# B&R Automation Studio project acopos6d_issues
Automation Studio 6.5.3.11; technology packages: mapp6D 3.6.0, mappConnect 6.1.0, mappSafety 6.0.0, mappServices 6.6.0, mappView 6.6.0, OpcUaCs 6.6.0

## Configuration Big

CPU 5APC4100.TGL2-000, AutomationRuntime 6.6.2, Build 11.3.0

### Task classes (Cpu.sw)
```
Cyclic#1 (cycle 2000 us, tolerance 0 us):
  Main <- src.Main.Main.prg
  FastDemo <- src.FastDemo.FastDemo.prg
Cyclic#2 (cycle 10000 us, tolerance 10000 us):
  Power <- src.Power.Power.prg
NcDataObjects: McDriveLog
Binaries: ArSvcReg, udbdef, FWRules, TCData, User, ashwac, iomap, UaCsConfig, sysconf, asfw, arconfig, BRRole, ashwd, Layout, Config_1, Config_2, McAcpDrv, mvLoader, Acp10map, acp10cfg, Settings, mCoWebSc, Config_4, Config_3, Config_8, Config_6, Config_7, Config_5
Libraries: operator, runtime, AsIecCon, astime, AsZip, FileIO, SegFind, Mover, AsBrMath, AsBrStr, brsystem, AsIODiag, sys_lib, AsTCP, standard, MpBase, McAcp6D, McBase, BrdkPackML, brdkSTR, PackMLCore, UaCore, McAcp6DSys, UaCoal, UaCoalPrv, powerlnk, AsEPL, ArSsl, MpTraffic, FastLib, SfDomain
```

### Hardware
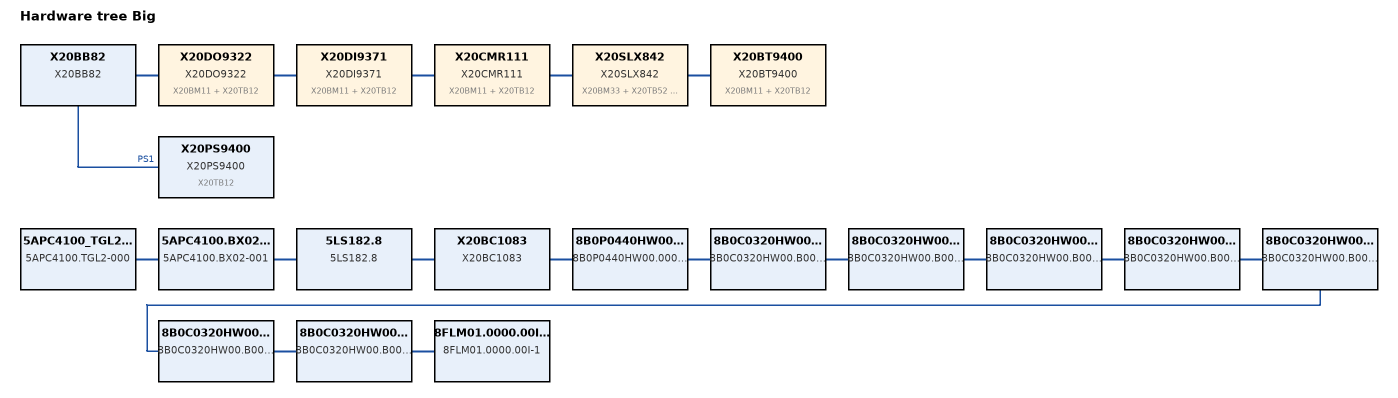
```
5APC4100.BX02-001 : 5APC4100.BX02-001 v1.0.0.0  [SY -> 5APC4100_TGL2_000.SY3]
5APC4100_TGL2_000 : 5APC4100.TGL2-000 v1.3.1.0
  Connector IF3:
    AssignedOperatingSystem = ARemb
    ActivateDevice = 1
    HostName = big-6d
    Mode = Manual
    InternetAddress = 192.168.1.101
    SubnetMask = 255.255.255.0
    ActivateSnmp = 2
  Connector IF4:
    AssignedOperatingSystem = ARemb
    ActivateDevice = 1
  Connector IF5:
    AssignedOperatingSystem = GPOS
  Connector IF6:
    AssignedOperatingSystem = GPOS
  Connector IF13:
    OperatingSystem = ARemb
    ActivateDevice = 1
  Connector IF7:
    AssignedOperatingSystem = GPOS
  Connector IF8:
    AssignedOperatingSystem = GPOS
  Connector IF9:
    AssignedOperatingSystem = GPOS
  Connector IF10:
    AssignedOperatingSystem = GPOS
  Connector IF11:
    AssignedOperatingSystem = ARemb
  Connector IF12:
    AssignedOperatingSystem = ARemb
  ConfigurationID = MainSystem_Config1
  ActivateHypervisor = 1
  ARembDramSizeInMb = 2048
  Simulation = 1
  TimerDeviceType = EPLX2X
  TimerDevice = 5LS182.8.IF1
  TaskClassIdleTime = 2000
  Cyclic1Duration = 2000
  Cyclic1Tolerance = 0
  Cyclic2Duration = 10000
  Cyclic2Tolerance = 10000
  FileDevice1
  FileDeviceName1 = 6DData
  FileDevicePath1 = USER_PATH
  ActivateFtpServer = 1
  FTPProtocol = 1
  FtpUser1
  FtpUsername1 = admin
  FtpUserPassword1 = xLRKj1BlFM98w2szVE2MiBEx5VuiwEUy/nukFErU7QU=
  FtpUserSalt1 = /uIGmoS1
  FTPAccessRight1 = 0
  FTPdevice1 = ALL
  ActivateWebServer = 1
  WebServerProtocol = 1
  ActivateSdm = 1
5LS182.8 : 5LS182.8 v1.5.1.0  [SL -> 5APC4100.BX02-001.SL1]
  Connector IF1:
    EplNatSubnet = 192.168.102.0
  Supervision = off
8B0C0320HW00.B00-1_A : 8B0C0320HW00.B00-1 v1.0.1.3 (NodeNumber=3)  [PLK1 -> 8B0P0440HW00.000-1.PLK2 [Cable Type=PowerlinkCable, Length=10, Version=1.0.0.3]; PLK2 -> 8B0C0320HW00.B00-1_B.PLK1 [Cable Type=PowerlinkCable, Length=10, Version=1.0.0.3]]
  FunctionModel = DirectControl
  Supervision = off
  OutputVoltage = 48000
  CurrentLimitation = Used
  OutputCurrentLimit = 20000
  OutputCurrentLimitTime = 20
  ConfigOutputState = off
8B0C0320HW00.B00-1_B : 8B0C0320HW00.B00-1 v1.0.1.3 (NodeNumber=4)  [PLK1 -> 8B0C0320HW00.B00-1_A.PLK2 [Cable Type=PowerlinkCable, Length=10, Version=1.0.0.3]; PLK2 -> 8B0C0320HW00.B00-1_C.PLK1 [Cable Type=PowerlinkCable, Length=10, Version=1.0.0.3]]
  FunctionModel = DirectControl
  Supervision = off
  OutputVoltage = 48000
  CurrentLimitation = Used
  OutputCurrentLimit = 20000
  OutputCurrentLimitTime = 20
  ConfigOutputState = off
8B0C0320HW00.B00-1_C : 8B0C0320HW00.B00-1 v1.0.1.3 (NodeNumber=5)  [PLK1 -> 8B0C0320HW00.B00-1_B.PLK2 [Cable Type=PowerlinkCable, Length=10, Version=1.0.0.3]; PLK2 -> 8B0C0320HW00.B00-1_D.PLK1 [Cable Type=PowerlinkCable, Length=10, Version=1.0.0.3]]
  FunctionModel = DirectControl
  Supervision = off
  OutputVoltage = 48000
  CurrentLimitation = Used
  OutputCurrentLimit = 20000
  OutputCurrentLimitTime = 20
  ConfigOutputState = off
8B0C0320HW00.B00-1_D : 8B0C0320HW00.B00-1 v1.0.1.3 (NodeNumber=6)  [PLK1 -> 8B0C0320HW00.B00-1_C.PLK2 [Cable Type=PowerlinkCable, Length=10, Version=1.0.0.3]; PLK2 -> 8B0C0320HW00.B00-1_E.PLK1 [Cable Type=PowerlinkCable, Length=10, Version=1.0.0.3]]
  FunctionModel = DirectControl
  Supervision = off
  OutputVoltage = 48000
  CurrentLimitation = Used
  OutputCurrentLimit = 20000
  OutputCurrentLimitTime = 20
  ConfigOutputState = off
8B0C0320HW00.B00-1_E : 8B0C0320HW00.B00-1 v1.0.1.3 (NodeNumber=7)  [PLK1 -> 8B0C0320HW00.B00-1_D.PLK2 [Cable Type=PowerlinkCable, Length=10, Version=1.0.0.3]; PLK2 -> 8B0C0320HW00.B00-1_F.PLK1 [Cable Type=PowerlinkCable, Length=10, Version=1.0.0.3]]
  FunctionModel = DirectControl
  Supervision = off
  OutputVoltage = 48000
  CurrentLimitation = Used
  OutputCurrentLimit = 20000
  OutputCurrentLimitTime = 20
  ConfigOutputState = off
8B0C0320HW00.B00-1_F : 8B0C0320HW00.B00-1 v1.0.1.3 (NodeNumber=8)  [PLK1 -> 8B0C0320HW00.B00-1_E.PLK2 [Cable Type=PowerlinkCable, Length=10, Version=1.0.0.3]; PLK2 -> 8B0C0320HW00.B00-1_G.PLK1 [Cable Type=PowerlinkCable, Length=10, Version=1.0.0.3]]
  FunctionModel = DirectControl
  Supervision = off
  OutputVoltage = 48000
  CurrentLimitation = Used
  OutputCurrentLimit = 20000
  OutputCurrentLimitTime = 20
  ConfigOutputState = off
8B0C0320HW00.B00-1_G : 8B0C0320HW00.B00-1 v1.0.1.3 (NodeNumber=9)  [PLK1 -> 8B0C0320HW00.B00-1_F.PLK2 [Cable Type=PowerlinkCable, Length=10, Version=1.0.0.3]; PLK2 -> 8FLM01.0000.00I-1.PLK1 [Cable Type=PowerlinkCable, Length=10, Version=1.0.0.3]]
  FunctionModel = DirectControl
  Supervision = off
  OutputVoltage = 48000
  CurrentLimitation = Used
  OutputCurrentLimit = 20000
  OutputCurrentLimitTime = 20
  ConfigOutputState = off
8B0P0440HW00.000-1 : 8B0P0440HW00.000-1 v2.3.0.3 (NodeNumber=2)  [PLK1 -> X20BC1083.PLK2 [Cable Type=PowerlinkCable, Length=10, Version=1.0.0.3]; PLK2 -> 8B0C0320HW00.B00-1_A.PLK1 [Cable Type=PowerlinkCable, Length=10, Version=1.0.0.3]]
  MotionTP = Acp10Arnc0
8FLM01.0000.00I-1 : 8FLM01.0000.00I-1 v1.0.0.2  [PLK1 -> 8B0C0320HW00.B00-1_G.PLK2 [Cable Type=PowerlinkCable, Length=10, Version=1.0.0.3]]
  Supervision = off
X20BB82 : X20BB82 v1.2.0.0
X20BC1083 : X20BC1083 v2.17.0.0 (NodeNumber=1)  [PLK1 -> 5LS182.8.IF1 [Cable Type=PowerlinkCable, Length=10, Version=1.0.0.3]; PLK2 -> 8B0P0440HW00.000-1.PLK1 [Cable Type=PowerlinkCable, Length=10, Version=1.0.0.3]; SL -> X20BB82.SL1]
  Supervision = off
X20BM11 : X20BM11 v1.1.0.0  [X2X1 -> X20BB82.IF1]
X20BM11_a : X20BM11 v1.1.0.0  [X2X1 -> X20BM11.X2X2]
X20BM11_b : X20BM11 v1.1.0.0  [X2X1 -> X20BM11_a.X2X2]
X20BM11_c : X20BM11 v1.1.0.0  [X2X1 -> X20BM33.X2X2]
X20BM33 : X20BM33 v1.1.0.0  [X2X1 -> X20BM11_b.X2X2]
X20BT9400 : X20BT9400 v1.4.0.0  [SS1 -> X20TB12_d.SS; SL -> X20BM11_c.SL1]
  Supervision = off
X20CMR111 : X20CMR111 v1.7.0.0  [SS1 -> X20TB12_c.SS; SL -> X20BM11_b.SL1]
  Supervision = off
X20DI9371 : X20DI9371 v1.6.1.0  [SS1 -> X20TB12_b.SS; SL -> X20BM11_a.SL1]
  Supervision = off
X20DO9322 : X20DO9322 v1.7.0.0  [SS1 -> X20TB12_a.SS; SL -> X20BM11.SL1]
  Supervision = off
X20PS9400 : X20PS9400 v1.9.0.0  [SS1 -> X20TB12.SS; PS -> X20BB82.PS1]
  Supervision = off
X20SLX842 : X20SLX842 v2.6.1.0  [SS1 -> X20TB52.SS; SS2 -> X20TB52_a.SS; SL -> X20BM33.SL1]
  Supervision = off
X20TB12 : X20TB12 v1.0.0.0
X20TB12_a : X20TB12 v1.0.0.0
X20TB12_b : X20TB12 v1.0.0.0
X20TB12_c : X20TB12 v1.0.0.0
X20TB12_d : X20TB12 v1.0.0.0
X20TB52 : X20TB52 v1.0.0.2
X20TB52_a : X20TB52 v1.0.0.2
```

### IoMap.iom - 5APC4100_TGL2_000/IoMap.iom
```iecst
VAR_CONFIG
	Cyclic#1.::gCommInput.Array[0] AT %IW."8FLM01.0000.00I-1".EPL_FB_IN_0_I2007_S01;
	Cyclic#1.::gCommInput.Array[1] AT %IW."8FLM01.0000.00I-1".EPL_FB_IN_1_I2007_S02;
	Cyclic#1.::gCommInput.Array[2] AT %IW."8FLM01.0000.00I-1".EPL_FB_IN_2_I2007_S03;
	Cyclic#1.::gCommInput.Array[3] AT %IW."8FLM01.0000.00I-1".EPL_FB_IN_3_I2007_S04;
	Cyclic#1.::gCommInput.Array[4] AT %IW."8FLM01.0000.00I-1".EPL_FB_IN_4_I2007_S05;
	Cyclic#1.::gCommInput.Array[5] AT %IW."8FLM01.0000.00I-1".EPL_FB_IN_5_I2007_S06;
	Cyclic#1.::gCommInput.Array[6] AT %IW."8FLM01.0000.00I-1".EPL_FB_IN_6_I2007_S07;
	Cyclic#1.::gCommInput.Array[7] AT %IW."8FLM01.0000.00I-1".EPL_FB_IN_7_I2007_S08;
	Cyclic#1.::gCommInput.Array[8] AT %IW."8FLM01.0000.00I-1".EPL_FB_IN_8_I2007_S09;
	Cyclic#1.::gCommInput.Array[9] AT %IW."8FLM01.0000.00I-1".EPL_FB_IN_9_I2007_S0A;
	Cyclic#1.::gCommInput.Array[10] AT %IW."8FLM01.0000.00I-1".EPL_FB_IN_10_I2007_S0B;
	Cyclic#1.::gCommInput.Array[11] AT %IW."8FLM01.0000.00I-1".EPL_FB_IN_11_I2007_S0C;
	Cyclic#1.::gCommInput.Array[12] AT %IW."8FLM01.0000.00I-1".EPL_FB_IN_12_I2007_S0D;
	Cyclic#1.::gCommInput.Array[13] AT %IW."8FLM01.0000.00I-1".EPL_FB_IN_13_I2007_S0E;
	Cyclic#1.::gCommInput.Array[14] AT %IW."8FLM01.0000.00I-1".EPL_FB_IN_14_I2007_S0F;
	Cyclic#1.::gCommInput.Array[15] AT %IW."8FLM01.0000.00I-1".EPL_FB_IN_15_I2007_S10;
	Cyclic#1.::gCommInput.Array[16] AT %IW."8FLM01.0000.00I-1".EPL_FB_IN_16_I2007_S11;
	Cyclic#1.::gCommInput.Array[17] AT %IW."8FLM01.0000.00I-1".EPL_FB_IN_17_I2007_S12;
	Cyclic#1.::gCommInput.Array[18] AT %IW."8FLM01.0000.00I-1".EPL_FB_IN_18_I2007_S13;
	Cyclic#1.::gCommInput.Array[19] AT %IW."8FLM01.0000.00I-1".EPL_FB_IN_19_I2007_S14;
	Cyclic#1.::gCommInput.Array[20] AT %IW."8FLM01.0000.00I-1".EPL_FB_IN_20_I2007_S15;
	Cyclic#1.::gCommInput.Array[21] AT %IW."8FLM01.0000.00I-1".EPL_FB_IN_21_I2007_S16;
	Cyclic#1.::gCommInput.Array[22] AT %IW."8FLM01.0000.00I-1".EPL_FB_IN_22_I2007_S17;
	Cyclic#1.::gCommInput.Array[23] AT %IW."8FLM01.0000.00I-1".EPL_FB_IN_23_I2007_S18;
	Cyclic#1.::gCommInput.Array[24] AT %IW."8FLM01.0000.00I-1".EPL_FB_IN_24_I2007_S19;
	Cyclic#1.::gCommInput.Array[25] AT %IW."8FLM01.0000.00I-1".EPL_FB_IN_25_I2007_S1A;
	Cyclic#1.::gCommInput.Array[26] AT %IW."8FLM01.0000.00I-1".EPL_FB_IN_26_I2007_S1B;
	Cyclic#1.::gCommInput.Array[27] AT %IW."8FLM01.0000.00I-1".EPL_FB_IN_27_I2007_S1C;
	Cyclic#1.::gCommInput.Array[28] AT %IW."8FLM01.0000.00I-1".EPL_FB_IN_28_I2007_S1D;
	Cyclic#1.::gCommInput.Array[29] AT %IW."8FLM01.0000.00I-1".EPL_FB_IN_29_I2007_S1E;
	Cyclic#1.::gCommInput.Array[30] AT %IW."8FLM01.0000.00I-1".EPL_FB_IN_30_I2007_S1F;
	Cyclic#1.::gCommInput.Array[31] AT %IW."8FLM01.0000.00I-1".EPL_FB_IN_31_I2007_S20;
	Cyclic#1.::gCommInput.Array[32] AT %IW."8FLM01.0000.00I-1".EPL_FB_IN_32_I2007_S21;
	Cyclic#1.::gCommInput.Array[33] AT %IW."8FLM01.0000.00I-1".EPL_FB_IN_33_I2007_S22;
	Cyclic#1.::gCommInput.Array[34] AT %IW."8FLM01.0000.00I-1".EPL_FB_IN_34_I2007_S23;
	Cyclic#1.::gCommInput.Array[35] AT %IW."8FLM01.0000.00I-1".EPL_FB_IN_35_I2007_S24;
	Cyclic#1.::gCommInput.Array[36] AT %IW."8FLM01.0000.00I-1".EPL_FB_IN_36_I2007_S25;
	Cyclic#1.::gCommInput.Array[37] AT %IW."8FLM01.0000.00I-1".EPL_FB_IN_37_I2007_S26;
	Cyclic#1.::gCommInput.Array[38] AT %IW."8FLM01.0000.00I-1".EPL_FB_IN_38_I2007_S27;
	Cyclic#1.::gCommInput.Array[39] AT %IW."8FLM01.0000.00I-1".EPL_FB_IN_39_I2007_S28;
	Cyclic#1.::gCommInput.Array[40] AT %IW."8FLM01.0000.00I-1".EPL_FB_IN_40_I2007_S29;
	Cyclic#1.::gCommInput.Array[41] AT %IW."8FLM01.0000.00I-1".EPL_FB_IN_41_I2007_S2A;
	Cyclic#1.::gCommInput.Array[42] AT %IW."8FLM01.0000.00I-1".EPL_FB_IN_42_I2007_S2B;
	Cyclic#1.::gCommInput.Array[43] AT %IW."8FLM01.0000.00I-1".EPL_FB_IN_43_I2007_S2C;
	Cyclic#1.::gCommInput.Array[44] AT %IW."8FLM01.0000.00I-1".EPL_FB_IN_44_I2007_S2D;
	Cyclic#1.::gCommInput.Array[45] AT %IW."8FLM01.0000.00I-1".EPL_FB_IN_45_I2007_S2E;
	Cyclic#1.::gCommInput.Array[46] AT %IW."8FLM01.0000.00I-1".EPL_FB_IN_46_I2007_S2F;
	Cyclic#1.::gCommInput.Array[47] AT %IW."8FLM01.0000.00I-1".EPL_FB_IN_47_I2007_S30;
	Cyclic#1.::gCommInput.Array[48] AT %IW."8FLM01.0000.00I-1".EPL_FB_IN_48_I2007_S31;
	Cyclic#1.::gCommInput.Array[49] AT %IW."8FLM01.0000.00I-1".EPL_FB_IN_49_I2007_S32;
	Cyclic#1.::gCommInput.Array[50] AT %IW."8FLM01.0000.00I-1".EPL_FB_IN_50_I2007_S33;
	Cyclic#1.::gCommInput.Array[51] AT %IW."8FLM01.0000.00I-1".EPL_FB_IN_51_I2007_S34;
	Cyclic#1.::gCommInput.Array[52] AT %IW."8FLM01.0000.00I-1".EPL_FB_IN_52_I2007_S35;
	Cyclic#1.::gCommInput.Array[53] AT %IW."8FLM01.0000.00I-1".EPL_FB_IN_53_I2007_S36;
	Cyclic#1.::gCommInput.Array[54] AT %IW."8FLM01.0000.00I-1".EPL_FB_IN_54_I2007_S37;
	Cyclic#1.::gCommInput.Array[55] AT %IW."8FLM01.0000.00I-1".EPL_FB_IN_55_I2007_S38;
	Cyclic#1.::gCommInput.Array[56] AT %IW."8FLM01.0000.00I-1".EPL_FB_IN_56_I2007_S39;
	Cyclic#1.::gCommInput.Array[57] AT %IW."8FLM01.0000.00I-1".EPL_FB_IN_57_I2007_S3A;
	Cyclic#1.::gCommInput.Array[58] AT %IW."8FLM01.0000.00I-1".EPL_FB_IN_58_I2007_S3B;
	Cyclic#1.::gCommInput.Array[59] AT %IW."8FLM01.0000.00I-1".EPL_FB_IN_59_I2007_S3C;
	Cyclic#1.::gCommInput.Array[60] AT %IW."8FLM01.0000.00I-1".EPL_FB_IN_60_I2007_S3D;
	Cyclic#1.::gCommInput.Array[61] AT %IW."8FLM01.0000.00I-1".EPL_FB_IN_61_I2007_S3E;
	Cyclic#1.::gCommInput.Array[62] AT %IW."8FLM01.0000.00I-1".EPL_FB_IN_62_I2007_S3F;
	Cyclic#1.::gCommInput.Array[63] AT %IW."8FLM01.0000.00I-1".EPL_FB_IN_63_I2007_S40;
	Cyclic#1.::gCommInput.Array[64] AT %IW."8FLM01.0000.00I-1".EPL_FB_IN_64_I2007_S41;
	Cyclic#1.::gCommInput.Array[65] AT %IW."8FLM01.0000.00I-1".EPL_FB_IN_65_I2007_S42;
	Cyclic#1.::gCommInput.Array[66] AT %IW."8FLM01.0000.00I-1".EPL_FB_IN_66_I2007_S43;
	Cyclic#1.::gCommInput.Array[67] AT %IW."8FLM01.0000.00I-1".EPL_FB_IN_67_I2007_S44;
	Cyclic#1.::gCommInput.Array[68] AT %IW."8FLM01.0000.00I-1".EPL_FB_IN_68_I2007_S45;
	Cyclic#1.::gCommInput.Array[69] AT %IW."8FLM01.0000.00I-1".EPL_FB_IN_69_I2007_S46;
	Cyclic#1.::gCommInput.Array[70] AT %IW."8FLM01.0000.00I-1".EPL_FB_IN_70_I2007_S47;
	Cyclic#1.::gCommInput.Array[71] AT %IW."8FLM01.0000.00I-1".EPL_FB_IN_71_I2007_S48;
	Cyclic#1.::gCommInput.Array[72] AT %IW."8FLM01.0000.00I-1".EPL_FB_IN_72_I2007_S49;
	Cyclic#1.::gCommInput.Array[73] AT %IW."8FLM01.0000.00I-1".EPL_FB_IN_73_I2007_S4A;
	Cyclic#1.::gCommInput.Array[74] AT %IW."8FLM01.0000.00I-1".EPL_FB_IN_74_I2007_S4B;
	Cyclic#1.::gCommInput.Array[75] AT %IW."8FLM01.0000.00I-1".EPL_FB_IN_75_I2007_S4C;
	Cyclic#1.::gCommInput.Array[76] AT %IW."8FLM01.0000.00I-1".EPL_FB_IN_76_I2007_S4D;
	Cyclic#1.::gCommInput.Array[77] AT %IW."8FLM01.0000.00I-1".EPL_FB_IN_77_I2007_S4E;
	Cyclic#1.::gCommInput.Array[78] AT %IW."8FLM01.0000.00I-1".EPL_FB_IN_78_I2007_S4F;
	Cyclic#1.::gCommInput.Array[79] AT %IW."8FLM01.0000.00I-1".EPL_FB_IN_79_I2007_S50;
	Cyclic#1.::gCommInput.Array[80] AT %IW."8FLM01.0000.00I-1".EPL_FB_IN_80_I2007_S51;
	Cyclic#1.::gCommInput.Array[81] AT %IW."8FLM01.0000.00I-1".EPL_FB_IN_81_I2007_S52;
	Cyclic#1.::gCommInput.Array[82] AT %IW."8FLM01.0000.00I-1".EPL_FB_IN_82_I2007_S53;
	Cyclic#1.::gCommInput.Array[83] AT %IW."8FLM01.0000.00I-1".EPL_FB_IN_83_I2007_S54;
	Cyclic#1.::gCommInput.Array[84] AT %IW."8FLM01.0000.00I-1".EPL_FB_IN_84_I2007_S55;
	Cyclic#1.::gCommInput.Array[85] AT %IW."8FLM01.0000.00I-1".EPL_FB_IN_85_I2007_S56;
	Cyclic#1.::gCommInput.Array[86] AT %IW."8FLM01.0000.00I-1".EPL_FB_IN_86_I2007_S57;
	Cyclic#1.::gCommInput.Array[87] AT %IW."8FLM01.0000.00I-1".EPL_FB_IN_87_I2007_S58;
	Cyclic#1.::gCommInput.Array[88] AT %IW."8FLM01.0000.00I-1".EPL_FB_IN_88_I2007_S59;
	Cyclic#1.::gCommInput.Array[89] AT %IW."8FLM01.0000.00I-1".EPL_FB_IN_89_I2007_S5A;
	Cyclic#1.::gCommInput.Array[90] AT %IW."8FLM01.0000.00I-1".EPL_FB_IN_90_I2007_S5B;
	Cyclic#1.::gCommInput.Array[91] AT %IW."8FLM01.0000.00I-1".EPL_FB_IN_91_I2007_S5C;
	Cyclic#1.::gCommInput.Array[92] AT %IW."8FLM01.0000.00I-1".EPL_FB_IN_92_I2007_S5D;
	Cyclic#1.::gCommInput.Array[93] AT %IW."8FLM01.0000.00I-1".EPL_FB_IN_93_I2007_S5E;
	Cyclic#1.::gCommInput.Array[94] AT %IW."8FLM01.0000.00I-1".EPL_FB_IN_94_I2007_S5F;
	Cyclic#1.::gCommInput.Array[95] AT %IW."8FLM01.0000.00I-1".EPL_FB_IN_95_I2007_S60;
	Cyclic#1.::gCommInput.Array[96] AT %IW."8FLM01.0000.00I-1".EPL_FB_IN_96_I2007_S61;
	Cyclic#1.::gCommInput.Array[97] AT %IW."8FLM01.0000.00I-1".EPL_FB_IN_97_I2007_S62;
	Cyclic#1.::gCommInput.Array[98] AT %IW."8FLM01.0000.00I-1".EPL_FB_IN_98_I2007_S63;
	Cyclic#1.::gCommInput.Array[99] AT %IW."8FLM01.0000.00I-1".EPL_FB_IN_99_I2007_S64;
	Cyclic#1.::gCommInput.Array[100] AT %IW."8FLM01.0000.00I-1".EPL_FB_IN_100_I2007_S65;
	Cyclic#1.::gCommInput.Array[101] AT %IW."8FLM01.0000.00I-1".EPL_FB_IN_101_I2007_S66;
	Cyclic#1.::gCommInput.Array[102] AT %IW."8FLM01.0000.00I-1".EPL_FB_IN_102_I2007_S67;
	Cyclic#1.::gCommInput.Array[103] AT %IW."8FLM01.0000.00I-1".EPL_FB_IN_103_I2007_S68;
	Cyclic#1.::gCommInput.Array[104] AT %IW."8FLM01.0000.00I-1".EPL_FB_IN_104_I2007_S69;
	Cyclic#1.::gCommInput.Array[105] AT %IW."8FLM01.0000.00I-1".EPL_FB_IN_105_I2007_S6A;
	Cyclic#1.::gCommInput.Array[106] AT %IW."8FLM01.0000.00I-1".EPL_FB_IN_106_I2007_S6B;
	Cyclic#1.::gCommInput.Array[107] AT %IW."8FLM01.0000.00I-1".EPL_FB_IN_107_I2007_S6C;
	Cyclic#1.::gCommInput.Array[108] AT %IW."8FLM01.0000.00I-1".EPL_FB_IN_108_I2007_S6D;
	Cyclic#1.::gCommInput.Array[109] AT %IW."8FLM01.0000.00I-1".EPL_FB_IN_109_I2007_S6E;
	Cyclic#1.::gCommInput.Array[110] AT %IW."8FLM01.0000.00I-1".EPL_FB_IN_110_I2007_S6F;
	Cyclic#1.::gCommInput.Array[111] AT %IW."8FLM01.0000.00I-1".EPL_FB_IN_111_I2007_S70;
	Cyclic#1.::gCommInput.Array[112] AT %IW."8FLM01.0000.00I-1".EPL_FB_IN_112_I2007_S71;
	Cyclic#1.::gCommInput.Array[113] AT %IW."8FLM01.0000.00I-1".EPL_FB_IN_113_I2007_S72;
	Cyclic#1.::gCommInput.Array[114] AT %IW."8FLM01.0000.00I-1".EPL_FB_IN_114_I2007_S73;
	Cyclic#1.::gCommInput.Array[115] AT %IW."8FLM01.0000.00I-1".EPL_FB_IN_115_I2007_S74;
	Cyclic#1.::gCommInput.Array[116] AT %IW."8FLM01.0000.00I-1".EPL_FB_IN_116_I2007_S75;
	Cyclic#1.::gCommInput.Array[117] AT %IW."8FLM01.0000.00I-1".EPL_FB_IN_117_I2007_S76;
	Cyclic#1.::gCommInput.Array[118] AT %IW."8FLM01.0000.00I-1".EPL_FB_IN_118_I2007_S77;
	Cyclic#1.::gCommInput.Array[119] AT %IW."8FLM01.0000.00I-1".EPL_FB_IN_119_I2007_S78;
	Cyclic#1.::gCommInput.Array[120] AT %IW."8FLM01.0000.00I-1".EPL_FB_IN_120_I2007_S79;
	Cyclic#1.::gCommInput.Array[121] AT %IW."8FLM01.0000.00I-1".EPL_FB_IN_121_I2007_S7A;
	Cyclic#1.::gCommInput.Array[122] AT %IW."8FLM01.0000.00I-1".EPL_FB_IN_122_I2007_S7B;
	Cyclic#1.::gCommInput.Array[123] AT %IW."8FLM01.0000.00I-1".EPL_FB_IN_123_I2007_S7C;
	Cyclic#1.::gCommInput.Array[124] AT %IW."8FLM01.0000.00I-1".EPL_FB_IN_124_I2007_S7D;
	Cyclic#1.::gCommInput.Array[125] AT %IW."8FLM01.0000.00I-1".EPL_FB_IN_125_I2007_S7E;
	Cyclic#1.::gCommInput.Array[126] AT %IW."8FLM01.0000.00I-1".EPL_FB_IN_126_I2007_S7F;
	Cyclic#1.::gCommInput.Array[127] AT %IW."8FLM01.0000.00I-1".EPL_FB_IN_127_I2007_S80;
	Cyclic#1.::gCommInput.Array[128] AT %IW."8FLM01.0000.00I-1".EPL_FB_IN_128_I2007_S81;
	Cyclic#1.::gCommInput.Array[129] AT %IW."8FLM01.0000.00I-1".EPL_FB_IN_129_I2007_S82;
	Cyclic#1.::gCommInput.Array[130] AT %IW."8FLM01.0000.00I-1".EPL_FB_IN_130_I2007_S83;
	Cyclic#1.::gCommInput.Array[131] AT %IW."8FLM01.0000.00I-1".EPL_FB_IN_131_I2007_S84;
	Cyclic#1.::gCommInput.Array[132] AT %IW."8FLM01.0000.00I-1".EPL_FB_IN_132_I2007_S85;
	Cyclic#1.::gCommInput.Array[133] AT %IW."8FLM01.0000.00I-1".EPL_FB_IN_133_I2007_S86;
	Cyclic#1.::gCommInput.Array[134] AT %IW."8FLM01.0000.00I-1".EPL_FB_IN_134_I2007_S87;
	Cyclic#1.::gCommInput.Array[135] AT %IW."8FLM01.0000.00I-1".EPL_FB_IN_135_I2007_S88;
	Cyclic#1.::gCommInput.Array[136] AT %IW."8FLM01.0000.00I-1".EPL_FB_IN_136_I2007_S89;
	Cyclic#1.::gCommInput.Array[137] AT %IW."8FLM01.0000.00I-1".EPL_FB_IN_137_I2007_S8A;
	Cyclic#1.::gCommInput.Array[138] AT %IW."8FLM01.0000.00I-1".EPL_FB_IN_138_I2007_S8B;
	Cyclic#1.::gCommInput.Array[139] AT %IW."8FLM01.0000.00I-1".EPL_FB_IN_139_I2007_S8C;
	Cyclic#1.::gCommInput.Array[140] AT %IW."8FLM01.0000.00I-1".EPL_FB_IN_140_I2007_S8D;
	Cyclic#1.::gCommInput.Array[141] AT %IW."8FLM01.0000.00I-1".EPL_FB_IN_141_I2007_S8E;
	Cyclic#1.::gCommInput.Array[142] AT %IW."8FLM01.0000.00I-1".EPL_FB_IN_142_I2007_S8F;
	Cyclic#1.::gCommInput.Array[143] AT %IW."8FLM01.0000.00I-1".EPL_FB_IN_143_I2007_S90;
	Cyclic#1.::gCommInput.Array[144] AT %IW."8FLM01.0000.00I-1".EPL_FB_IN_144_I2007_S91;
	Cyclic#1.::gCommInput.Array[145] AT %IW."8FLM01.0000.00I-1".EPL_FB_IN_145_I2007_S92;
	Cyclic#1.::gCommInput.Array[146] AT %IW."8FLM01.0000.00I-1".EPL_FB_IN_146_I2007_S93;
	Cyclic#1.::gCommInput.Array[147] AT %IW."8FLM01.0000.00I-1".EPL_FB_IN_147_I2007_S94;
	Cyclic#1.::gCommInput.Array[148] AT %IW."8FLM01.0000.00I-1".EPL_FB_IN_148_I2007_S95;
	Cyclic#1.::gCommInput.Array[149] AT %IW."8FLM01.0000.00I-1".EPL_FB_IN_149_I2007_S96;
	Cyclic#1.::gCommInput.Array[150] AT %IW."8FLM01.0000.00I-1".EPL_FB_IN_150_I2007_S97;
	Cyclic#1.::gCommInput.Array[151] AT %IW."8FLM01.0000.00I-1".EPL_FB_IN_151_I2007_S98;
	Cyclic#1.::gCommInput.Array[152] AT %IW."8FLM01.0000.00I-1".EPL_FB_IN_152_I2007_S99;
	Cyclic#1.::gCommInput.Array[153] AT %IW."8FLM01.0000.00I-1".EPL_FB_IN_153_I2007_S9A;
	Cyclic#1.::gCommInput.Array[154] AT %IW."8FLM01.0000.00I-1".EPL_FB_IN_154_I2007_S9B;
	Cyclic#1.::gCommInput.Array[155] AT %IW."8FLM01.0000.00I-1".EPL_FB_IN_155_I2007_S9C;
	Cyclic#1.::gCommInput.Array[156] AT %IW."8FLM01.0000.00I-1".EPL_FB_IN_156_I2007_S9D;
	Cyclic#1.::gCommInput.Array[157] AT %IW."8FLM01.0000.00I-1".EPL_FB_IN_157_I2007_S9E;
	Cyclic#1.::gCommInput.Array[158] AT %IW."8FLM01.0000.00I-1".EPL_FB_IN_158_I2007_S9F;
	Cyclic#1.::gCommInput.Array[159] AT %IW."8FLM01.0000.00I-1".EPL_FB_IN_159_I2007_SA0;
	Cyclic#1.::gCommInput.Array[160] AT %IW."8FLM01.0000.00I-1".EPL_FB_IN_160_I2007_SA1;
	Cyclic#1.::gCommInput.Array[161] AT %IW."8FLM01.0000.00I-1".EPL_FB_IN_161_I2007_SA2;
	Cyclic#1.::gCommInput.Array[162] AT %IW."8FLM01.0000.00I-1".EPL_FB_IN_162_I2007_SA3;
	Cyclic#1.::gCommInput.Array[163] AT %IW."8FLM01.0000.00I-1".EPL_FB_IN_163_I2007_SA4;
	Cyclic#1.::gCommInput.Array[164] AT %IW."8FLM01.0000.00I-1".EPL_FB_IN_164_I2007_SA5;
	Cyclic#1.::gCommInput.Array[165] AT %IW."8FLM01.0000.00I-1".EPL_FB_IN_165_I2007_SA6;
	Cyclic#1.::gCommInput.Array[166] AT %IW."8FLM01.0000.00I-1".EPL_FB_IN_166_I2007_SA7;
	Cyclic#1.::gCommInput.Array[167] AT %IW."8FLM01.0000.00I-1".EPL_FB_IN_167_I2007_SA8;
	Cyclic#1.::gCommInput.Array[168] AT %IW."8FLM01.0000.00I-1".EPL_FB_IN_168_I2007_SA9;
	Cyclic#1.::gCommInput.Array[169] AT %IW."8FLM01.0000.00I-1".EPL_FB_IN_169_I2007_SAA;
	Cyclic#1.::gCommInput.Array[170] AT %IW."8FLM01.0000.00I-1".EPL_FB_IN_170_I2007_SAB;
	Cyclic#1.::gCommInput.Array[171] AT %IW."8FLM01.0000.00I-1".EPL_FB_IN_171_I2007_SAC;
	Cyclic#1.::gCommInput.Array[172] AT %IW."8FLM01.0000.00I-1".EPL_FB_IN_172_I2007_SAD;
	Cyclic#1.::gCommInput.Array[173] AT %IW."8FLM01.0000.00I-1".EPL_FB_IN_173_I2007_SAE;
	Cyclic#1.::gCommInput.Array[174] AT %IW."8FLM01.0000.00I-1".EPL_FB_IN_174_I2007_SAF;
	Cyclic#1.::gCommInput.Array[175] AT %IW."8FLM01.0000.00I-1".EPL_FB_IN_175_I2007_SB0;
	Cyclic#1.::gCommInput.Array[176] AT %IW."8FLM01.0000.00I-1".EPL_FB_IN_176_I2007_SB1;
	Cyclic#1.::gCommInput.Array[177] AT %IW."8FLM01.0000.00I-1".EPL_FB_IN_177_I2007_SB2;
	Cyclic#1.::gCommInput.Array[178] AT %IW."8FLM01.0000.00I-1".EPL_FB_IN_178_I2007_SB3;
	Cyclic#1.::gCommInput.Array[179] AT %IW."8FLM01.0000.00I-1".EPL_FB_IN_179_I2007_SB4;
	Cyclic#1.::gCommInput.Array[180] AT %IW."8FLM01.0000.00I-1".EPL_FB_IN_180_I2007_SB5;
	Cyclic#1.::gCommInput.Array[181] AT %IW."8FLM01.0000.00I-1".EPL_FB_IN_181_I2007_SB6;
	Cyclic#1.::gCommInput.Array[182] AT %IW."8FLM01.0000.00I-1".EPL_FB_IN_182_I2007_SB7;
	Cyclic#1.::gCommInput.Array[183] AT %IW."8FLM01.0000.00I-1".EPL_FB_IN_183_I2007_SB8;
	Cyclic#1.::gCommInput.Array[184] AT %IW."8FLM01.0000.00I-1".EPL_FB_IN_184_I2007_SB9;
	Cyclic#1.::gCommInput.Array[185] AT %IW."8FLM01.0000.00I-1".EPL_FB_IN_185_I2007_SBA;
	Cyclic#1.::gCommInput.Array[186] AT %IW."8FLM01.0000.00I-1".EPL_FB_IN_186_I2007_SBB;
	Cyclic#1.::gCommInput.Array[187] AT %IW."8FLM01.0000.00I-1".EPL_FB_IN_187_I2007_SBC;
	Cyclic#1.::gCommInput.Array[188] AT %IW."8FLM01.0000.00I-1".EPL_FB_IN_188_I2007_SBD;
	Cyclic#1.::gCommInput.Array[189] AT %IW."8FLM01.0000.00I-1".EPL_FB_IN_189_I2007_SBE;
	Cyclic#1.::gCommInput.Array[190] AT %IW."8FLM01.0000.00I-1".EPL_FB_IN_190_I2007_SBF;
	Cyclic#1.::gCommInput.Array[191] AT %IW."8FLM01.0000.00I-1".EPL_FB_IN_191_I2007_SC0;
	Cyclic#1.::gCommInput.Array[192] AT %IW."8FLM01.0000.00I-1".EPL_FB_IN_192_I2007_SC1;
	Cyclic#1.::gCommInput.Array[193] AT %IW."8FLM01.0000.00I-1".EPL_FB_IN_193_I2007_SC2;
	Cyclic#1.::gCommInput.Array[194] AT %IW."8FLM01.0000.00I-1".EPL_FB_IN_194_I2007_SC3;
	Cyclic#1.::gCommInput.Array[195] AT %IW."8FLM01.0000.00I-1".EPL_FB_IN_195_I2007_SC4;
	Cyclic#1.::gCommInput.Array[196] AT %IW."8FLM01.0000.00I-1".EPL_FB_IN_196_I2007_SC5;
	Cyclic#1.::gCommInput.Array[197] AT %IW."8FLM01.0000.00I-1".EPL_FB_IN_197_I2007_SC6;
	Cyclic#1.::gCommInput.Array[198] AT %IW."8FLM01.0000.00I-1".EPL_FB_IN_198_I2007_SC7;
	Cyclic#1.::gCommInput.Array[199] AT %IW."8FLM01.0000.00I-1".EPL_FB_IN_199_I2007_SC8;
	Cyclic#1.::gCommOutput.Array[0] AT %QW."8FLM01.0000.00I-1".EPL_FB_OUT_0_I2008_S01Out;
	Cyclic#1.::gCommOutput.Array[1] AT %QW."8FLM01.0000.00I-1".EPL_FB_OUT_1_I2008_S02Out;
	Cyclic#1.::gCommOutput.Array[2] AT %QW."8FLM01.0000.00I-1".EPL_FB_OUT_2_I2008_S03Out;
	Cyclic#1.::gCommOutput.Array[3] AT %QW."8FLM01.0000.00I-1".EPL_FB_OUT_3_I2008_S04Out;
	Cyclic#1.::gCommOutput.Array[4] AT %QW."8FLM01.0000.00I-1".EPL_FB_OUT_4_I2008_S05Out;
	Cyclic#1.::gCommOutput.Array[5] AT %QW."8FLM01.0000.00I-1".EPL_FB_OUT_5_I2008_S06Out;
	Cyclic#1.::gCommOutput.Array[6] AT %QW."8FLM01.0000.00I-1".EPL_FB_OUT_6_I2008_S07Out;
	Cyclic#1.::gCommOutput.Array[7] AT %QW."8FLM01.0000.00I-1".EPL_FB_OUT_7_I2008_S08Out;
	Cyclic#1.::gCommOutput.Array[8] AT %QW."8FLM01.0000.00I-1".EPL_FB_OUT_8_I2008_S09Out;
	Cyclic#1.::gCommOutput.Array[9] AT %QW."8FLM01.0000.00I-1".EPL_FB_OUT_9_I2008_S0AOut;
	Cyclic#1.::gCommOutput.Array[10] AT %QW."8FLM01.0000.00I-1".EPL_FB_OUT_10_I2008_S0BOut;
	Cyclic#1.::gCommOutput.Array[11] AT %QW."8FLM01.0000.00I-1".EPL_FB_OUT_11_I2008_S0COut;
	Cyclic#1.::gCommOutput.Array[12] AT %QW."8FLM01.0000.00I-1".EPL_FB_OUT_12_I2008_S0DOut;
	Cyclic#1.::gCommOutput.Array[13] AT %QW."8FLM01.0000.00I-1".EPL_FB_OUT_13_I2008_S0EOut;
	Cyclic#1.::gCommOutput.Array[14] AT %QW."8FLM01.0000.00I-1".EPL_FB_OUT_14_I2008_S0FOut;
	Cyclic#1.::gCommOutput.Array[15] AT %QW."8FLM01.0000.00I-1".EPL_FB_OUT_15_I2008_S10Out;
	Cyclic#1.::gCommOutput.Array[16] AT %QW."8FLM01.0000.00I-1".EPL_FB_OUT_16_I2008_S11Out;
	Cyclic#1.::gCommOutput.Array[17] AT %QW."8FLM01.0000.00I-1".EPL_FB_OUT_17_I2008_S12Out;
	Cyclic#1.::gCommOutput.Array[18] AT %QW."8FLM01.0000.00I-1".EPL_FB_OUT_18_I2008_S13Out;
	Cyclic#1.::gCommOutput.Array[19] AT %QW."8FLM01.0000.00I-1".EPL_FB_OUT_19_I2008_S14Out;
	Cyclic#1.::gCommOutput.Array[20] AT %QW."8FLM01.0000.00I-1".EPL_FB_OUT_20_I2008_S15Out;
	Cyclic#1.::gCommOutput.Array[21] AT %QW."8FLM01.0000.00I-1".EPL_FB_OUT_21_I2008_S16Out;
	Cyclic#1.::gCommOutput.Array[22] AT %QW."8FLM01.0000.00I-1".EPL_FB_OUT_22_I2008_S17Out;
	Cyclic#1.::gCommOutput.Array[23] AT %QW."8FLM01.0000.00I-1".EPL_FB_OUT_23_I2008_S18Out;
	Cyclic#1.::gCommOutput.Array[24] AT %QW."8FLM01.0000.00I-1".EPL_FB_OUT_24_I2008_S19Out;
	Cyclic#1.::gCommOutput.Array[25] AT %QW."8FLM01.0000.00I-1".EPL_FB_OUT_25_I2008_S1AOut;
	Cyclic#1.::gCommOutput.Array[26] AT %QW."8FLM01.0000.00I-1".EPL_FB_OUT_26_I2008_S1BOut;
	Cyclic#1.::gCommOutput.Array[27] AT %QW."8FLM01.0000.00I-1".EPL_FB_OUT_27_I2008_S1COut;
	Cyclic#1.::gCommOutput.Array[28] AT %QW."8FLM01.0000.00I-1".EPL_FB_OUT_28_I2008_S1DOut;
	Cyclic#1.::gCommOutput.Array[29] AT %QW."8FLM01.0000.00I-1".EPL_FB_OUT_29_I2008_S1EOut;
	Cyclic#1.::gCommOutput.Array[30] AT %QW."8FLM01.0000.00I-1".EPL_FB_OUT_30_I2008_S1FOut;
	Cyclic#1.::gCommOutput.Array[31] AT %QW."8FLM01.0000.00I-1".EPL_FB_OUT_31_I2008_S20Out;
	Cyclic#1.::gCommOutput.Array[32] AT %QW."8FLM01.0000.00I-1".EPL_FB_OUT_32_I2008_S21Out;
	Cyclic#1.::gCommOutput.Array[33] AT %QW."8FLM01.0000.00I-1".EPL_FB_OUT_33_I2008_S22Out;
	Cyclic#1.::gCommOutput.Array[34] AT %QW."8FLM01.0000.00I-1".EPL_FB_OUT_34_I2008_S23Out;
	Cyclic#1.::gCommOutput.Array[35] AT %QW."8FLM01.0000.00I-1".EPL_FB_OUT_35_I2008_S24Out;
	Cyclic#1.::gCommOutput.Array[36] AT %QW."8FLM01.0000.00I-1".EPL_FB_OUT_36_I2008_S25Out;
	Cyclic#1.::gCommOutput.Array[37] AT %QW."8FLM01.0000.00I-1".EPL_FB_OUT_37_I2008_S26Out;
	Cyclic#1.::gCommOutput.Array[38] AT %QW."8FLM01.0000.00I-1".EPL_FB_OUT_38_I2008_S27Out;
	Cyclic#1.::gCommOutput.Array[39] AT %QW."8FLM01.0000.00I-1".EPL_FB_OUT_39_I2008_S28Out;
	Cyclic#1.::gCommOutput.Array[40] AT %QW."8FLM01.0000.00I-1".EPL_FB_OUT_40_I2008_S29Out;
	Cyclic#1.::gCommOutput.Array[41] AT %QW."8FLM01.0000.00I-1".EPL_FB_OUT_41_I2008_S2AOut;
	Cyclic#1.::gCommOutput.Array[42] AT %QW."8FLM01.0000.00I-1".EPL_FB_OUT_42_I2008_S2BOut;
	Cyclic#1.::gCommOutput.Array[43] AT %QW."8FLM01.0000.00I-1".EPL_FB_OUT_43_I2008_S2COut;
	Cyclic#1.::gCommOutput.Array[44] AT %QW."8FLM01.0000.00I-1".EPL_FB_OUT_44_I2008_S2DOut;
	Cyclic#1.::gCommOutput.Array[45] AT %QW."8FLM01.0000.00I-1".EPL_FB_OUT_45_I2008_S2EOut;
	Cyclic#1.::gCommOutput.Array[46] AT %QW."8FLM01.0000.00I-1".EPL_FB_OUT_46_I2008_S2FOut;
	Cyclic#1.::gCommOutput.Array[47] AT %QW."8FLM01.0000.00I-1".EPL_FB_OUT_47_I2008_S30Out;
	Cyclic#1.::gCommOutput.Array[48] AT %QW."8FLM01.0000.00I-1".EPL_FB_OUT_48_I2008_S31Out;
	Cyclic#1.::gCommOutput.Array[49] AT %QW."8FLM01.0000.00I-1".EPL_FB_OUT_49_I2008_S32Out;
	Cyclic#1.::gCommOutput.Array[50] AT %QW."8FLM01.0000.00I-1".EPL_FB_OUT_50_I2008_S33Out;
	Cyclic#1.::gCommOutput.Array[51] AT %QW."8FLM01.0000.00I-1".EPL_FB_OUT_51_I2008_S34Out;
	Cyclic#1.::gCommOutput.Array[52] AT %QW."8FLM01.0000.00I-1".EPL_FB_OUT_52_I2008_S35Out;
	Cyclic#1.::gCommOutput.Array[53] AT %QW."8FLM01.0000.00I-1".EPL_FB_OUT_53_I2008_S36Out;
	Cyclic#1.::gCommOutput.Array[54] AT %QW."8FLM01.0000.00I-1".EPL_FB_OUT_54_I2008_S37Out;
	Cyclic#1.::gCommOutput.Array[55] AT %QW."8FLM01.0000.00I-1".EPL_FB_OUT_55_I2008_S38Out;
	Cyclic#1.::gCommOutput.Array[56] AT %QW."8FLM01.0000.00I-1".EPL_FB_OUT_56_I2008_S39Out;
	Cyclic#1.::gCommOutput.Array[57] AT %QW."8FLM01.0000.00I-1".EPL_FB_OUT_57_I2008_S3AOut;
	Cyclic#1.::gCommOutput.Array[58] AT %QW."8FLM01.0000.00I-1".EPL_FB_OUT_58_I2008_S3BOut;
	Cyclic#1.::gCommOutput.Array[59] AT %QW."8FLM01.0000.00I-1".EPL_FB_OUT_59_I2008_S3COut;
	Cyclic#1.::gCommOutput.Array[60] AT %QW."8FLM01.0000.00I-1".EPL_FB_OUT_60_I2008_S3DOut;
	Cyclic#1.::gCommOutput.Array[61] AT %QW."8FLM01.0000.00I-1".EPL_FB_OUT_61_I2008_S3EOut;
	Cyclic#1.::gCommOutput.Array[62] AT %QW."8FLM01.0000.00I-1".EPL_FB_OUT_62_I2008_S3FOut;
	Cyclic#1.::gCommOutput.Array[63] AT %QW."8FLM01.0000.00I-1".EPL_FB_OUT_63_I2008_S40Out;
	Cyclic#1.::gCommOutput.Array[64] AT %QW."8FLM01.0000.00I-1".EPL_FB_OUT_64_I2008_S41Out;
	Cyclic#1.::gCommOutput.Array[65] AT %QW."8FLM01.0000.00I-1".EPL_FB_OUT_65_I2008_S42Out;
	Cyclic#1.::gCommOutput.Array[66] AT %QW."8FLM01.0000.00I-1".EPL_FB_OUT_66_I2008_S43Out;
	Cyclic#1.::gCommOutput.Array[67] AT %QW."8FLM01.0000.00I-1".EPL_FB_OUT_67_I2008_S44Out;
	Cyclic#1.::gCommOutput.Array[68] AT %QW."8FLM01.0000.00I-1".EPL_FB_OUT_68_I2008_S45Out;
	Cyclic#1.::gCommOutput.Array[69] AT %QW."8FLM01.0000.00I-1".EPL_FB_OUT_69_I2008_S46Out;
	Cyclic#1.::gCommOutput.Array[70] AT %QW."8FLM01.0000.00I-1".EPL_FB_OUT_70_I2008_S47Out;
	Cyclic#1.::gCommOutput.Array[71] AT %QW."8FLM01.0000.00I-1".EPL_FB_OUT_71_I2008_S48Out;
	Cyclic#1.::gCommOutput.Array[72] AT %QW."8FLM01.0000.00I-1".EPL_FB_OUT_72_I2008_S49Out;
	Cyclic#1.::gCommOutput.Array[73] AT %QW."8FLM01.0000.00I-1".EPL_FB_OUT_73_I2008_S4AOut;
	Cyclic#1.::gCommOutput.Array[74] AT %QW."8FLM01.0000.00I-1".EPL_FB_OUT_74_I2008_S4BOut;
	Cyclic#1.::gCommOutput.Array[75] AT %QW."8FLM01.0000.00I-1".EPL_FB_OUT_75_I2008_S4COut;
	Cyclic#1.::gCommOutput.Array[76] AT %QW."8FLM01.0000.00I-1".EPL_FB_OUT_76_I2008_S4DOut;
	Cyclic#1.::gCommOutput.Array[77] AT %QW."8FLM01.0000.00I-1".EPL_FB_OUT_77_I2008_S4EOut;
	Cyclic#1.::gCommOutput.Array[78] AT %QW."8FLM01.0000.00I-1".EPL_FB_OUT_78_I2008_S4FOut;
	Cyclic#1.::gCommOutput.Array[79] AT %QW."8FLM01.0000.00I-1".EPL_FB_OUT_79_I2008_S50Out;
	Cyclic#1.::gCommOutput.Array[80] AT %QW."8FLM01.0000.00I-1".EPL_FB_OUT_80_I2008_S51Out;
	Cyclic#1.::gCommOutput.Array[81] AT %QW."8FLM01.0000.00I-1".EPL_FB_OUT_81_I2008_S52Out;
	Cyclic#1.::gCommOutput.Array[82] AT %QW."8FLM01.0000.00I-1".EPL_FB_OUT_82_I2008_S53Out;
	Cyclic#1.::gCommOutput.Array[83] AT %QW."8FLM01.0000.00I-1".EPL_FB_OUT_83_I2008_S54Out;
	Cyclic#1.::gCommOutput.Array[84] AT %QW."8FLM01.0000.00I-1".EPL_FB_OUT_84_I2008_S55Out;
	Cyclic#1.::gCommOutput.Array[85] AT %QW."8FLM01.0000.00I-1".EPL_FB_OUT_85_I2008_S56Out;
	Cyclic#1.::gCommOutput.Array[86] AT %QW."8FLM01.0000.00I-1".EPL_FB_OUT_86_I2008_S57Out;
	Cyclic#1.::gCommOutput.Array[87] AT %QW."8FLM01.0000.00I-1".EPL_FB_OUT_87_I2008_S58Out;
	Cyclic#1.::gCommOutput.Array[88] AT %QW."8FLM01.0000.00I-1".EPL_FB_OUT_88_I2008_S59Out;
	Cyclic#1.::gCommOutput.Array[89] AT %QW."8FLM01.0000.00I-1".EPL_FB_OUT_89_I2008_S5AOut;
	Cyclic#1.::gCommOutput.Array[90] AT %QW."8FLM01.0000.00I-1".EPL_FB_OUT_90_I2008_S5BOut;
	Cyclic#1.::gCommOutput.Array[91] AT %QW."8FLM01.0000.00I-1".EPL_FB_OUT_91_I2008_S5COut;
	Cyclic#1.::gCommOutput.Array[92] AT %QW."8FLM01.0000.00I-1".EPL_FB_OUT_92_I2008_S5DOut;
	Cyclic#1.::gCommOutput.Array[93] AT %QW."8FLM01.0000.00I-1".EPL_FB_OUT_93_I2008_S5EOut;
	Cyclic#1.::gCommOutput.Array[94] AT %QW."8FLM01.0000.00I-1".EPL_FB_OUT_94_I2008_S5FOut;
	Cyclic#1.::gCommOutput.Array[95] AT %QW."8FLM01.0000.00I-1".EPL_FB_OUT_95_I2008_S60Out;
	Cyclic#1.::gCommOutput.Array[96] AT %QW."8FLM01.0000.00I-1".EPL_FB_OUT_96_I2008_S61Out;
	Cyclic#1.::gCommOutput.Array[97] AT %QW."8FLM01.0000.00I-1".EPL_FB_OUT_97_I2008_S62Out;
	Cyclic#1.::gCommOutput.Array[98] AT %QW."8FLM01.0000.00I-1".EPL_FB_OUT_98_I2008_S63Out;
	Cyclic#1.::gCommOutput.Array[99] AT %QW."8FLM01.0000.00I-1".EPL_FB_OUT_99_I2008_S64Out;
	Cyclic#1.::gCommOutput.Array[100] AT %QW."8FLM01.0000.00I-1".EPL_FB_OUT_100_I2008_S65Out;
	Cyclic#1.::gCommOutput.Array[101] AT %QW."8FLM01.0000.00I-1".EPL_FB_OUT_101_I2008_S66Out;
	Cyclic#1.::gCommOutput.Array[102] AT %QW."8FLM01.0000.00I-1".EPL_FB_OUT_102_I2008_S67Out;
	Cyclic#1.::gCommOutput.Array[103] AT %QW."8FLM01.0000.00I-1".EPL_FB_OUT_103_I2008_S68Out;
	Cyclic#1.::gCommOutput.Array[104] AT %QW."8FLM01.0000.00I-1".EPL_FB_OUT_104_I2008_S69Out;
	Cyclic#1.::gCommOutput.Array[105] AT %QW."8FLM01.0000.00I-1".EPL_FB_OUT_105_I2008_S6AOut;
	Cyclic#1.::gCommOutput.Array[106] AT %QW."8FLM01.0000.00I-1".EPL_FB_OUT_106_I2008_S6BOut;
	Cyclic#1.::gCommOutput.Array[107] AT %QW."8FLM01.0000.00I-1".EPL_FB_OUT_107_I2008_S6COut;
	Cyclic#1.::gCommOutput.Array[108] AT %QW."8FLM01.0000.00I-1".EPL_FB_OUT_108_I2008_S6DOut;
	Cyclic#1.::gCommOutput.Array[109] AT %QW."8FLM01.0000.00I-1".EPL_FB_OUT_109_I2008_S6EOut;
	Cyclic#1.::gCommOutput.Array[110] AT %QW."8FLM01.0000.00I-1".EPL_FB_OUT_110_I2008_S6FOut;
	Cyclic#1.::gCommOutput.Array[111] AT %QW."8FLM01.0000.00I-1".EPL_FB_OUT_111_I2008_S70Out;
	Cyclic#1.::gCommOutput.Array[112] AT %QW."8FLM01.0000.00I-1".EPL_FB_OUT_112_I2008_S71Out;
	Cyclic#1.::gCommOutput.Array[113] AT %QW."8FLM01.0000.00I-1".EPL_FB_OUT_113_I2008_S72Out;
	Cyclic#1.::gCommOutput.Array[114] AT %QW."8FLM01.0000.00I-1".EPL_FB_OUT_114_I2008_S73Out;
	Cyclic#1.::gCommOutput.Array[115] AT %QW."8FLM01.0000.00I-1".EPL_FB_OUT_115_I2008_S74Out;
	Cyclic#1.::gCommOutput.Array[116] AT %QW."8FLM01.0000.00I-1".EPL_FB_OUT_116_I2008_S75Out;
	Cyclic#1.::gCommOutput.Array[117] AT %QW."8FLM01.0000.00I-1".EPL_FB_OUT_117_I2008_S76Out;
	Cyclic#1.::gCommOutput.Array[118] AT %QW."8FLM01.0000.00I-1".EPL_FB_OUT_118_I2008_S77Out;
	Cyclic#1.::gCommOutput.Array[119] AT %QW."8FLM01.0000.00I-1".EPL_FB_OUT_119_I2008_S78Out;
	Cyclic#1.::gCommOutput.Array[120] AT %QW."8FLM01.0000.00I-1".EPL_FB_OUT_120_I2008_S79Out;
	Cyclic#1.::gCommOutput.Array[121] AT %QW."8FLM01.0000.00I-1".EPL_FB_OUT_121_I2008_S7AOut;
	Cyclic#1.::gCommOutput.Array[122] AT %QW."8FLM01.0000.00I-1".EPL_FB_OUT_122_I2008_S7BOut;
	Cyclic#1.::gCommOutput.Array[123] AT %QW."8FLM01.0000.00I-1".EPL_FB_OUT_123_I2008_S7COut;
	Cyclic#1.::gCommOutput.Array[124] AT %QW."8FLM01.0000.00I-1".EPL_FB_OUT_124_I2008_S7DOut;
	Cyclic#1.::gCommOutput.Array[125] AT %QW."8FLM01.0000.00I-1".EPL_FB_OUT_125_I2008_S7EOut;
	Cyclic#1.::gCommOutput.Array[126] AT %QW."8FLM01.0000.00I-1".EPL_FB_OUT_126_I2008_S7FOut;
	Cyclic#1.::gCommOutput.Array[127] AT %QW."8FLM01.0000.00I-1".EPL_FB_OUT_127_I2008_S80Out;
	Cyclic#1.::gCommOutput.Array[128] AT %QW."8FLM01.0000.00I-1".EPL_FB_OUT_128_I2008_S81Out;
	Cyclic#1.::gCommOutput.Array[129] AT %QW."8FLM01.0000.00I-1".EPL_FB_OUT_129_I2008_S82Out;
	Cyclic#1.::gCommOutput.Array[130] AT %QW."8FLM01.0000.00I-1".EPL_FB_OUT_130_I2008_S83Out;
	Cyclic#1.::gCommOutput.Array[131] AT %QW."8FLM01.0000.00I-1".EPL_FB_OUT_131_I2008_S84Out;
	Cyclic#1.::gCommOutput.Array[132] AT %QW."8FLM01.0000.00I-1".EPL_FB_OUT_132_I2008_S85Out;
	Cyclic#1.::gCommOutput.Array[133] AT %QW."8FLM01.0000.00I-1".EPL_FB_OUT_133_I2008_S86Out;
	Cyclic#1.::gCommOutput.Array[134] AT %QW."8FLM01.0000.00I-1".EPL_FB_OUT_134_I2008_S87Out;
	Cyclic#1.::gCommOutput.Array[135] AT %QW."8FLM01.0000.00I-1".EPL_FB_OUT_135_I2008_S88Out;
	Cyclic#1.::gCommOutput.Array[136] AT %QW."8FLM01.0000.00I-1".EPL_FB_OUT_136_I2008_S89Out;
	Cyclic#1.::gCommOutput.Array[137] AT %QW."8FLM01.0000.00I-1".EPL_FB_OUT_137_I2008_S8AOut;
	Cyclic#1.::gCommOutput.Array[138] AT %QW."8FLM01.0000.00I-1".EPL_FB_OUT_138_I2008_S8BOut;
	Cyclic#1.::gCommOutput.Array[139] AT %QW."8FLM01.0000.00I-1".EPL_FB_OUT_139_I2008_S8COut;
	Cyclic#1.::gCommOutput.Array[140] AT %QW."8FLM01.0000.00I-1".EPL_FB_OUT_140_I2008_S8DOut;
	Cyclic#1.::gCommOutput.Array[141] AT %QW."8FLM01.0000.00I-1".EPL_FB_OUT_141_I2008_S8EOut;
	Cyclic#1.::gCommOutput.Array[142] AT %QW."8FLM01.0000.00I-1".EPL_FB_OUT_142_I2008_S8FOut;
	Cyclic#1.::gCommOutput.Array[143] AT %QW."8FLM01.0000.00I-1".EPL_FB_OUT_143_I2008_S90Out;
	Cyclic#1.::gCommOutput.Array[144] AT %QW."8FLM01.0000.00I-1".EPL_FB_OUT_144_I2008_S91Out;
	Cyclic#1.::gCommOutput.Array[145] AT %QW."8FLM01.0000.00I-1".EPL_FB_OUT_145_I2008_S92Out;
	Cyclic#1.::gCommOutput.Array[146] AT %QW."8FLM01.0000.00I-1".EPL_FB_OUT_146_I2008_S93Out;
	Cyclic#1.::gCommOutput.Array[147] AT %QW."8FLM01.0000.00I-1".EPL_FB_OUT_147_I2008_S94Out;
	Cyclic#1.::gCommOutput.Array[148] AT %QW."8FLM01.0000.00I-1".EPL_FB_OUT_148_I2008_S95Out;
	Cyclic#1.::gCommOutput.Array[149] AT %QW."8FLM01.0000.00I-1".EPL_FB_OUT_149_I2008_S96Out;
	Cyclic#1.::gCommOutput.Array[150] AT %QW."8FLM01.0000.00I-1".EPL_FB_OUT_150_I2008_S97Out;
	Cyclic#1.::gCommOutput.Array[151] AT %QW."8FLM01.0000.00I-1".EPL_FB_OUT_151_I2008_S98Out;
	Cyclic#1.::gCommOutput.Array[152] AT %QW."8FLM01.0000.00I-1".EPL_FB_OUT_152_I2008_S99Out;
	Cyclic#1.::gCommOutput.Array[153] AT %QW."8FLM01.0000.00I-1".EPL_FB_OUT_153_I2008_S9AOut;
	Cyclic#1.::gCommOutput.Array[154] AT %QW."8FLM01.0000.00I-1".EPL_FB_OUT_154_I2008_S9BOut;
	Cyclic#1.::gCommOutput.Array[155] AT %QW."8FLM01.0000.00I-1".EPL_FB_OUT_155_I2008_S9COut;
	Cyclic#1.::gCommOutput.Array[156] AT %QW."8FLM01.0000.00I-1".EPL_FB_OUT_156_I2008_S9DOut;
	Cyclic#1.::gCommOutput.Array[157] AT %QW."8FLM01.0000.00I-1".EPL_FB_OUT_157_I2008_S9EOut;
	Cyclic#1.::gCommOutput.Array[158] AT %QW."8FLM01.0000.00I-1".EPL_FB_OUT_158_I2008_S9FOut;
	Cyclic#1.::gCommOutput.Array[159] AT %QW."8FLM01.0000.00I-1".EPL_FB_OUT_159_I2008_SA0Out;
	Cyclic#1.::gCommOutput.Array[160] AT %QW."8FLM01.0000.00I-1".EPL_FB_OUT_160_I2008_SA1Out;
	Cyclic#1.::gCommOutput.Array[161] AT %QW."8FLM01.0000.00I-1".EPL_FB_OUT_161_I2008_SA2Out;
	Cyclic#1.::gCommOutput.Array[162] AT %QW."8FLM01.0000.00I-1".EPL_FB_OUT_162_I2008_SA3Out;
	Cyclic#1.::gCommOutput.Array[163] AT %QW."8FLM01.0000.00I-1".EPL_FB_OUT_163_I2008_SA4Out;
	Cyclic#1.::gCommOutput.Array[164] AT %QW."8FLM01.0000.00I-1".EPL_FB_OUT_164_I2008_SA5Out;
	Cyclic#1.::gCommOutput.Array[165] AT %QW."8FLM01.0000.00I-1".EPL_FB_OUT_165_I2008_SA6Out;
	Cyclic#1.::gCommOutput.Array[166] AT %QW."8FLM01.0000.00I-1".EPL_FB_OUT_166_I2008_SA7Out;
	Cyclic#1.::gCommOutput.Array[167] AT %QW."8FLM01.0000.00I-1".EPL_FB_OUT_167_I2008_SA8Out;
	Cyclic#1.::gCommOutput.Array[168] AT %QW."8FLM01.0000.00I-1".EPL_FB_OUT_168_I2008_SA9Out;
	Cyclic#1.::gCommOutput.Array[169] AT %QW."8FLM01.0000.00I-1".EPL_FB_OUT_169_I2008_SAAOut;
	Cyclic#1.::gCommOutput.Array[170] AT %QW."8FLM01.0000.00I-1".EPL_FB_OUT_170_I2008_SABOut;
	Cyclic#1.::gCommOutput.Array[171] AT %QW."8FLM01.0000.00I-1".EPL_FB_OUT_171_I2008_SACOut;
	Cyclic#1.::gCommOutput.Array[172] AT %QW."8FLM01.0000.00I-1".EPL_FB_OUT_172_I2008_SADOut;
	Cyclic#1.::gCommOutput.Array[173] AT %QW."8FLM01.0000.00I-1".EPL_FB_OUT_173_I2008_SAEOut;
	Cyclic#1.::gCommOutput.Array[174] AT %QW."8FLM01.0000.00I-1".EPL_FB_OUT_174_I2008_SAFOut;
	Cyclic#1.::gCommOutput.Array[175] AT %QW."8FLM01.0000.00I-1".EPL_FB_OUT_175_I2008_SB0Out;
	Cyclic#1.::gCommOutput.Array[176] AT %QW."8FLM01.0000.00I-1".EPL_FB_OUT_176_I2008_SB1Out;
	Cyclic#1.::gCommOutput.Array[177] AT %QW."8FLM01.0000.00I-1".EPL_FB_OUT_177_I2008_SB2Out;
	Cyclic#1.::gCommOutput.Array[178] AT %QW."8FLM01.0000.00I-1".EPL_FB_OUT_178_I2008_SB3Out;
	Cyclic#1.::gCommOutput.Array[179] AT %QW."8FLM01.0000.00I-1".EPL_FB_OUT_179_I2008_SB4Out;
	Cyclic#1.::gCommOutput.Array[180] AT %QW."8FLM01.0000.00I-1".EPL_FB_OUT_180_I2008_SB5Out;
	Cyclic#1.::gCommOutput.Array[181] AT %QW."8FLM01.0000.00I-1".EPL_FB_OUT_181_I2008_SB6Out;
	Cyclic#1.::gCommOutput.Array[182] AT %QW."8FLM01.0000.00I-1".EPL_FB_OUT_182_I2008_SB7Out;
	Cyclic#1.::gCommOutput.Array[183] AT %QW."8FLM01.0000.00I-1".EPL_FB_OUT_183_I2008_SB8Out;
	Cyclic#1.::gCommOutput.Array[184] AT %QW."8FLM01.0000.00I-1".EPL_FB_OUT_184_I2008_SB9Out;
	Cyclic#1.::gCommOutput.Array[185] AT %QW."8FLM01.0000.00I-1".EPL_FB_OUT_185_I2008_SBAOut;
	Cyclic#1.::gCommOutput.Array[186] AT %QW."8FLM01.0000.00I-1".EPL_FB_OUT_186_I2008_SBBOut;
	Cyclic#1.::gCommOutput.Array[187] AT %QW."8FLM01.0000.00I-1".EPL_FB_OUT_187_I2008_SBCOut;
	Cyclic#1.::gCommOutput.Array[188] AT %QW."8FLM01.0000.00I-1".EPL_FB_OUT_188_I2008_SBDOut;
	Cyclic#1.::gCommOutput.Array[189] AT %QW."8FLM01.0000.00I-1".EPL_FB_OUT_189_I2008_SBEOut;
	Cyclic#1.::gCommOutput.Array[190] AT %QW."8FLM01.0000.00I-1".EPL_FB_OUT_190_I2008_SBFOut;
	Cyclic#1.::gCommOutput.Array[191] AT %QW."8FLM01.0000.00I-1".EPL_FB_OUT_191_I2008_SC0Out;
	Cyclic#1.::gCommOutput.Array[192] AT %QW."8FLM01.0000.00I-1".EPL_FB_OUT_192_I2008_SC1Out;
	Cyclic#1.::gCommOutput.Array[193] AT %QW."8FLM01.0000.00I-1".EPL_FB_OUT_193_I2008_SC2Out;
	Cyclic#1.::gCommOutput.Array[194] AT %QW."8FLM01.0000.00I-1".EPL_FB_OUT_194_I2008_SC3Out;
	Cyclic#1.::gCommOutput.Array[195] AT %QW."8FLM01.0000.00I-1".EPL_FB_OUT_195_I2008_SC4Out;
	Cyclic#1.::gCommOutput.Array[196] AT %QW."8FLM01.0000.00I-1".EPL_FB_OUT_196_I2008_SC5Out;
	Cyclic#1.::gCommOutput.Array[197] AT %QW."8FLM01.0000.00I-1".EPL_FB_OUT_197_I2008_SC6Out;
	Cyclic#1.::gCommOutput.Array[198] AT %QW."8FLM01.0000.00I-1".EPL_FB_OUT_198_I2008_SC7Out;
	Cyclic#1.::gCommOutput.Array[199] AT %QW."8FLM01.0000.00I-1".EPL_FB_OUT_199_I2008_SC8Out;
	::gPower.AuxPowerUnit[0].Command.EnableOutput AT %QX."8B0C0320HW00.B00-1_A".EnableOutput;
	::gPower.AuxPowerUnit[0].Command.DisableOutput AT %QX."8B0C0320HW00.B00-1_A".DisableOutput;
	::gPower.AuxPowerUnit[0].Command.AcknowledgeAllErrors AT %QX."8B0C0320HW00.B00-1_A".AcknowledgeAllErrors;
	::gPower.AuxPowerUnit[0].Command.AcknowledgeAllWarnings AT %QX."8B0C0320HW00.B00-1_A".AcknowledgeAllWarnings;
	::gPower.AuxPowerUnit[0].CrOk AT %IX."8B0C0320HW00.B00-1_A".CrOk;
	::gPower.AuxPowerUnit[0].OutputEnabled AT %IX."8B0C0320HW00.B00-1_A".OutputEnabled;
	::gPower.AuxPowerUnit[0].StatusRunMode AT %IB."8B0C0320HW00.B00-1_A".StatusRunMode;
	::gPower.AuxPowerUnit[0].Current_A AT %ID."8B0C0320HW00.B00-1_A".Iout;
	::gPower.AuxPowerUnit[0].Voltage_V AT %ID."8B0C0320HW00.B00-1_A".Uout;
	::gPower.AuxPowerUnit[1].Command.EnableOutput AT %QX."8B0C0320HW00.B00-1_B".EnableOutput;
	::gPower.AuxPowerUnit[1].Command.DisableOutput AT %QX."8B0C0320HW00.B00-1_B".DisableOutput;
	::gPower.AuxPowerUnit[1].Command.AcknowledgeAllErrors AT %QX."8B0C0320HW00.B00-1_B".AcknowledgeAllErrors;
	::gPower.AuxPowerUnit[1].Command.AcknowledgeAllWarnings AT %QX."8B0C0320HW00.B00-1_B".AcknowledgeAllWarnings;
	::gPower.AuxPowerUnit[1].CrOk AT %IX."8B0C0320HW00.B00-1_B".CrOk;
	::gPower.AuxPowerUnit[1].OutputEnabled AT %IX."8B0C0320HW00.B00-1_B".OutputEnabled;
	::gPower.AuxPowerUnit[1].StatusRunMode AT %IB."8B0C0320HW00.B00-1_B".StatusRunMode;
	::gPower.AuxPowerUnit[1].Current_A AT %ID."8B0C0320HW00.B00-1_B".Iout;
	::gPower.AuxPowerUnit[1].Voltage_V AT %ID."8B0C0320HW00.B00-1_B".Uout;
	::gPower.AuxPowerUnit[2].Command.EnableOutput AT %QX."8B0C0320HW00.B00-1_C".EnableOutput;
	::gPower.AuxPowerUnit[2].Command.DisableOutput AT %QX."8B0C0320HW00.B00-1_C".DisableOutput;
	::gPower.AuxPowerUnit[2].Command.AcknowledgeAllErrors AT %QX."8B0C0320HW00.B00-1_C".AcknowledgeAllErrors;
	::gPower.AuxPowerUnit[2].Command.AcknowledgeAllWarnings AT %QX."8B0C0320HW00.B00-1_C".AcknowledgeAllWarnings;
	::gPower.AuxPowerUnit[2].CrOk AT %IX."8B0C0320HW00.B00-1_C".CrOk;
	::gPower.AuxPowerUnit[2].OutputEnabled AT %IX."8B0C0320HW00.B00-1_C".OutputEnabled;
	::gPower.AuxPowerUnit[2].StatusRunMode AT %IB."8B0C0320HW00.B00-1_C".StatusRunMode;
	::gPower.AuxPowerUnit[2].Current_A AT %ID."8B0C0320HW00.B00-1_C".Iout;
	::gPower.AuxPowerUnit[2].Voltage_V AT %ID."8B0C0320HW00.B00-1_C".Uout;
	::gPower.AuxPowerUnit[3].Command.EnableOutput AT %QX."8B0C0320HW00.B00-1_D".EnableOutput;
	::gPower.AuxPowerUnit[3].Command.DisableOutput AT %QX."8B0C0320HW00.B00-1_D".DisableOutput;
	::gPower.AuxPowerUnit[3].Command.AcknowledgeAllErrors AT %QX."8B0C0320HW00.B00-1_D".AcknowledgeAllErrors;
	::gPower.AuxPowerUnit[3].Command.AcknowledgeAllWarnings AT %QX."8B0C0320HW00.B00-1_D".AcknowledgeAllWarnings;
	::gPower.AuxPowerUnit[3].CrOk AT %IX."8B0C0320HW00.B00-1_D".CrOk;
	::gPower.AuxPowerUnit[3].OutputEnabled AT %IX."8B0C0320HW00.B00-1_D".OutputEnabled;
	::gPower.AuxPowerUnit[3].StatusRunMode AT %IB."8B0C0320HW00.B00-1_D".StatusRunMode;
	::gPower.AuxPowerUnit[3].Current_A AT %ID."8B0C0320HW00.B00-1_D".Iout;
	::gPower.AuxPowerUnit[3].Voltage_V AT %ID."8B0C0320HW00.B00-1_D".Uout;
	::gPower.AuxPowerUnit[4].Command.EnableOutput AT %QX."8B0C0320HW00.B00-1_E".EnableOutput;
	::gPower.AuxPowerUnit[4].Command.DisableOutput AT %QX."8B0C0320HW00.B00-1_E".DisableOutput;
	::gPower.AuxPowerUnit[4].Command.AcknowledgeAllErrors AT %QX."8B0C0320HW00.B00-1_E".AcknowledgeAllErrors;
	::gPower.AuxPowerUnit[4].Command.AcknowledgeAllWarnings AT %QX."8B0C0320HW00.B00-1_E".AcknowledgeAllWarnings;
	::gPower.AuxPowerUnit[4].CrOk AT %IX."8B0C0320HW00.B00-1_E".CrOk;
	::gPower.AuxPowerUnit[4].OutputEnabled AT %IX."8B0C0320HW00.B00-1_E".OutputEnabled;
	::gPower.AuxPowerUnit[4].StatusRunMode AT %IB."8B0C0320HW00.B00-1_E".StatusRunMode;
	::gPower.AuxPowerUnit[4].Current_A AT %ID."8B0C0320HW00.B00-1_E".Iout;
	::gPower.AuxPowerUnit[4].Voltage_V AT %ID."8B0C0320HW00.B00-1_E".Uout;
	::gPower.AuxPowerUnit[5].Command.EnableOutput AT %QX."8B0C0320HW00.B00-1_F".EnableOutput;
	::gPower.AuxPowerUnit[5].Command.DisableOutput AT %QX."8B0C0320HW00.B00-1_F".DisableOutput;
	::gPower.AuxPowerUnit[5].Command.AcknowledgeAllErrors AT %QX."8B0C0320HW00.B00-1_F".AcknowledgeAllErrors;
	::gPower.AuxPowerUnit[5].Command.AcknowledgeAllWarnings AT %QX."8B0C0320HW00.B00-1_F".AcknowledgeAllWarnings;
	::gPower.AuxPowerUnit[5].CrOk AT %IX."8B0C0320HW00.B00-1_F".CrOk;
	::gPower.AuxPowerUnit[5].OutputEnabled AT %IX."8B0C0320HW00.B00-1_F".OutputEnabled;
	::gPower.AuxPowerUnit[5].StatusRunMode AT %IB."8B0C0320HW00.B00-1_F".StatusRunMode;
	::gPower.AuxPowerUnit[5].Current_A AT %ID."8B0C0320HW00.B00-1_F".Iout;
	::gPower.AuxPowerUnit[5].Voltage_V AT %ID."8B0C0320HW00.B00-1_F".Uout;
	::gPower.AuxPowerUnit[6].Command.EnableOutput AT %QX."8B0C0320HW00.B00-1_G".EnableOutput;
	::gPower.AuxPowerUnit[6].Command.DisableOutput AT %QX."8B0C0320HW00.B00-1_G".DisableOutput;
	::gPower.AuxPowerUnit[6].Command.AcknowledgeAllErrors AT %QX."8B0C0320HW00.B00-1_G".AcknowledgeAllErrors;
	::gPower.AuxPowerUnit[6].Command.AcknowledgeAllWarnings AT %QX."8B0C0320HW00.B00-1_G".AcknowledgeAllWarnings;
	::gPower.AuxPowerUnit[6].CrOk AT %IX."8B0C0320HW00.B00-1_G".CrOk;
	::gPower.AuxPowerUnit[6].OutputEnabled AT %IX."8B0C0320HW00.B00-1_G".OutputEnabled;
	::gPower.AuxPowerUnit[6].StatusRunMode AT %IB."8B0C0320HW00.B00-1_G".StatusRunMode;
	::gPower.AuxPowerUnit[6].Current_A AT %ID."8B0C0320HW00.B00-1_G".Iout;
	::gPower.AuxPowerUnit[6].Voltage_V AT %ID."8B0C0320HW00.B00-1_G".Uout;
	::gDI.Button1 AT %IX."X20DI9371".DigitalInput01;
	::gDI.Button2  AT %IX."X20DI9371".DigitalInput02;
	::gDI.Button3  AT %IX."X20DI9371".DigitalInput03;
	gDO.Button1_Led AT %QX."X20DO9322".DigitalOutput01;
	gDO.Button2_Led  AT %QX."X20DO9322".DigitalOutput02;
	gDO.Button3_Led  AT %QX."X20DO9322".DigitalOutput03;
END_VAR
```

### Config_2.trafficmanager - 5APC4100_TGL2_000/mapp6D/6DLaunchPad/TrafficManager_x6d_1/Config_2.trafficmanager
```
Element TrafficManager_x6d_1 (Type=trafficmanager)
  Base = AssemblyAcp6D
    BaseRef = gAssembly6D_Big
  TrafficObjects:
    TrafficObjectListRef[1] = Stations_1
    TrafficObjectListRef[2] = Waypoints_1
    TrafficObjectListRef[3] = Gates_1
  TrafficMapping:
    TrafficMappingListRef[1] = StationsMapping_1
    TrafficMappingListRef[2] = WaypointsMapping_1
    TrafficMappingListRef[3] = GatesMapping_1
  TrafficRules:
    TrafficRuleListRef[1] = Rules_1
  TrafficRecipes:
    TrafficRecipeRef[1] = Recipe_1
```

### Config_3.trafficobjectlist - 5APC4100_TGL2_000/mapp6D/6DLaunchPad/TrafficManager_x6d_1/Config_3.trafficobjectlist
```
Element Stations_1 (Type=trafficobjectlist)
  TrafficObject[1] = Station
    Name = S1
    Position = Absolute
      X = 0.3
      Y = 0.42
    RecoveryPoints:
      Mode = Direct
      StationIsRecoveryPoint = Enable
      RecoveryPoint[1]:
        Position = Absolute
          X = 0.3
          Y = 0.54
  TrafficObject[2] = Station
    Name = S2
    Position = Absolute
      X = 0.66
      Y = 0.06
    RecoveryPoints:
      Mode = Direct
      StationIsRecoveryPoint = Enable
  TrafficObject[3] = Station
    Name = S3
    Position = Absolute
      X = 0.66
      Y = 1.5
    RecoveryPoints:
      Mode = Direct
      StationIsRecoveryPoint = Enable
  TrafficObject[4] = Station
    Name = S4
    Position = Absolute
      X = 0.54
      Y = 1.5
    RecoveryPoints:
      Mode = Direct
      StationIsRecoveryPoint = Enable
  TrafficObject[5] = Station
    Name = S6
    Position = Absolute
      X = 0.66
      Y = 4.26
    RecoveryPoints:
      Mode = Direct
      StationIsRecoveryPoint = Enable
  TrafficObject[6] = Station
    Name = S5
    Position = Absolute
      X = 0.66
      Y = 2.94
    RecoveryPoints:
      Mode = Direct
      StationIsRecoveryPoint = Enable
  TrafficObject[7] = Station
    Name = S7
    Position = Absolute
      X = 0.3
      Y = 3.3
    RecoveryPoints:
      Mode = Direct
      StationIsRecoveryPoint = Enable
  TrafficObject[8] = Station
    Name = B1
    Position = Absolute
      X = 0.66
      Y = 1.38
    RecoveryPoints:
      Mode = Direct
      StationIsRecoveryPoint = Enable
  TrafficObject[9] = Station
    Name = B2
    Position = Absolute
      X = 0.3
      Y = 4.14
    RecoveryPoints:
      Mode = Direct
      StationIsRecoveryPoint = Enable
Element Waypoints_1 (Type=trafficobjectlist)
Element Gates_1 (Type=trafficobjectlist)
  TrafficObject[1] = Waypoint
    Name = G3
    Position = Absolute
      X = 0.66
      Y = 0.42
  TrafficObject[2] = Waypoint
    Name = G9
    Position = Absolute
      X = 0.42
      Y = 4.14
  TrafficObject[3] = Waypoint
    Name = G6
    Position = Absolute
      X = 0.54
      Y = 2.22
  TrafficObject[4] = Waypoint
    Name = G5
    Position = Absolute
      X = 0.66
      Y = 2.22
  TrafficObject[5] = Waypoint
    Name = G4
    Position = Absolute
      X = 0.66
      Y = 1.86
  TrafficObject[6] = Waypoint
    Name = G12
    Position = Absolute
      X = 0.3
      Y = 2.94
  TrafficObject[7] = Waypoint
    Name = G1
    Position = Absolute
      X = 0.3
      Y = 0.06
  TrafficObject[8] = Waypoint
    Name = G8
    Position = Absolute
      X = 0.66
      Y = 3.3
  TrafficObject[9] = Waypoint
    Name = G13
    Position = Absolute
      X = 0.54
      Y = 1.38
  TrafficObject[10] = Waypoint
    Name = G15
    Position = Absolute
      X = 0.42
      Y = 0.42
  TrafficObject[11] = Waypoint
    Name = G16
    Position = Absolute
      X = 0.3
      Y = 4.26
  TrafficObject[12] = Waypoint
    Name = G17
    Position = Absolute
      X = 0.54
      Y = 1.86
```

### Config_4.trafficmappinglist - 5APC4100_TGL2_000/mapp6D/6DLaunchPad/TrafficManager_x6d_1/Config_4.trafficmappinglist
```
Element StationsMapping_1 (Type=trafficmappinglist)
  TrafficMapping[1]:
    Source = Station
      SourceRef = S1
      Destinations:
        To[1] = Waypoint
          DestinationRef = G1
  TrafficMapping[2]:
    Source = Station
      SourceRef = S2
      Destinations:
        To[1] = Waypoint
          DestinationRef = G3
  TrafficMapping[3]:
    Source = Station
      SourceRef = S3
      Destinations:
        To[1] = Waypoint
          DestinationRef = G4
  TrafficMapping[4]:
    Source = Station
      SourceRef = S4
      Destinations:
        To[1] = Waypoint
          DestinationRef = G17
  TrafficMapping[5]:
    Source = Station
      SourceRef = S6
      Destinations:
        To[1] = Waypoint
          DestinationRef = G16
  TrafficMapping[6]:
    Source = Station
      SourceRef = S5
      Destinations:
        To[1] = Waypoint
          DestinationRef = G8
  TrafficMapping[7]:
    Source = Station
      SourceRef = S7
      Destinations:
        To[1] = Station
          DestinationRef = S1
  TrafficMapping[8]:
    Source = Station
      SourceRef = B1
      Destinations:
        To[1] = Station
          DestinationRef = S3
        To[2] = Waypoint
          DestinationRef = G13
  TrafficMapping[9]:
    Source = Station
      SourceRef = B2
      Destinations:
        To[1] = Station
          DestinationRef = S7
        To[2] = Waypoint
          DestinationRef = G9
Element WaypointsMapping_1 (Type=trafficmappinglist)
Element GatesMapping_1 (Type=trafficmappinglist)
  TrafficMapping[1]:
    Source = Waypoint
      SourceRef = G3
      Destinations:
        To[1] = Station
          DestinationRef = B1
  TrafficMapping[2]:
    Source = Waypoint
      SourceRef = G9
      Destinations:
        To[1] = Waypoint
          DestinationRef = G15
  TrafficMapping[3]:
    Source = Waypoint
      SourceRef = G6
      Destinations:
        To[1] = Waypoint
          DestinationRef = G5
  TrafficMapping[4]:
    Source = Waypoint
      SourceRef = G5
      Destinations:
        To[1] = Station
          DestinationRef = S5
  TrafficMapping[5]:
    Source = Waypoint
      SourceRef = G4
      Destinations:
        To[1] = Waypoint
          DestinationRef = G5
  TrafficMapping[6]:
    Source = Waypoint
      SourceRef = G1
      Destinations:
        To[1] = Station
          DestinationRef = S2
  TrafficMapping[7]:
    Source = Waypoint
      SourceRef = G8
      Destinations:
        To[1] = Station
          DestinationRef = S6
  TrafficMapping[8]:
    Source = Waypoint
      SourceRef = G13
      Destinations:
        To[1] = Station
          DestinationRef = S4
  TrafficMapping[9]:
    Source = Waypoint
      SourceRef = G15
      Destinations:
        To[1] = Station
          DestinationRef = S1
  TrafficMapping[10]:
    Source = Waypoint
      SourceRef = G16
      Destinations:
        To[1] = Station
          DestinationRef = B2
  TrafficMapping[11]:
    Source = Waypoint
      SourceRef = G17
      Destinations:
        To[1] = Waypoint
          DestinationRef = G6
```

### Config_5.trafficrulelist - 5APC4100_TGL2_000/mapp6D/6DLaunchPad/TrafficManager_x6d_1/Config_5.trafficrulelist
```
Element Rules_1 (Type=trafficrulelist)
  TrafficRule[1] = ExclusivityGroup
    Name = ExclusiveGroup_1
    TrafficObjects:
      TrafficObject[1] = Waypoint
        ExclusivityGroupObjectRef = G5
    EntryObjects
    ExitObjects
```

### Config_6.trafficrecipe - 5APC4100_TGL2_000/mapp6D/6DLaunchPad/TrafficManager_x6d_1/Config_6.trafficrecipe
```
Element Recipe_1 (Type=trafficrecipe)
  ProductLabel
  ProcessStep[1]:
    StationName = S1
    Process = DwellTime
      DwellTime = 1
    Transition = Next
      ToStation = S2
      Velocity = 2
      Acceleration = 18
  ProcessStep[2]:
    StationName = S2
    Process = DwellTime
      DwellTime = 1
    Transition = Next
      ToStation = B1
      Velocity = 2
      Acceleration = 18
  ProcessStep[3]:
    StationName = B1
    Process = DwellTime
      DwellTime = 0
    Transition = Distribution
      Branch[1]:
        ShuttleCount = 1
        ToStation = S3
        Velocity = 2
        Acceleration = 18
      Branch[2]:
        ShuttleCount = 1
        ToStation = S4
        Velocity = 2
        Acceleration = 18
  ProcessStep[4]:
    StationName = S3
    Process = DwellTime
      DwellTime = 1
    Transition = Next
      ToStation = S5
      Velocity = 2
      Acceleration = 18
  ProcessStep[5]:
    StationName = S4
    Process = DwellTime
      DwellTime = 1
    Transition = Next
      ToStation = S5
      Velocity = 2
      Acceleration = 18
  ProcessStep[6]:
    StationName = S5
    Process = DwellTime
      DwellTime = 1
    Transition = Next
      ToStation = S6
      Velocity = 2
      Acceleration = 18
  ProcessStep[7]:
    StationName = S6
    Process = DwellTime
      DwellTime = 1
    Transition = Next
      ToStation = B2
      Velocity = 2
      Acceleration = 18
  ProcessStep[8]:
    StationName = B2
    Process = DwellTime
      DwellTime = 0
    Transition = Distribution
      Branch[1]:
        ShuttleCount = 1
        ToStation = S7
        Velocity = 2
        Acceleration = 18
      Branch[2]:
        ShuttleCount = 1
        ToStation = S1
        Velocity = 2
        Acceleration = 18
  ProcessStep[9]:
    StationName = S7
    Process = DwellTime
      DwellTime = 1
    Transition = Next
      ToStation = S1
      Velocity = 2
      Acceleration = 18
```

### Asm6D.assembly6d - 5APC4100_TGL2_000/mapp6D/Asm6D.assembly6d
```
Element gAssembly6D_Big (Type=assembly6d)
  Simulation6D = SimOff
  Ethernet6D:
    IpAddress = 192.168.1.100
    SubnetMask = 255.255.255.0
    Gateway = 192.168.1.1
  Shuttles:
    MaxShuttleCount = 10  // Maximum count of shuttles in the assembly
    ShuttleIDMode = RealTimeID
    RealModeDetectionType = Any
    DefaultPosition:
      DefZ = 1.2
      DefRx = 0
      DefRy = 0
      DefRz = 0
    Limits:
      InPlaneLimits:
        InPlaneVelLim = 2.0
        InPlaneAccLim = 20
        InPlaneEmergDec = 20
      ShortAxLim:
        ShortAxAccLim:
          AccZLim = 10.0
          AccRxLim = 10.0
          AccRyLim = 10.0
          AccRzLim = 10.0
        ShortAxVelLim:
          VelZLim = 0.15
          VelRxLim = 0.1
          VelRyLim = 0.1
          VelRzLim = 0.1
    UserData:
      UserDataVariable
  CyclicChannel6D:
    ReadChannel:
      Xaxis = TRUE
      Yaxis = TRUE
      Zaxis = TRUE
      Rxaxis = TRUE
      Ryaxis = TRUE
      Rzaxis = TRUE
  SystemReactions6D:
    LostCommReaction6D = Continue
  Fieldbus6D:
    SyncMode6D = InternalSync
    IFName = SL1.IF1
    NodeNumber = 239
  IOMapp:
    Input = gCommInput
    Output = gCommOutput
  Layout:
    Layout6D[1] = Layout6D_Big
```

### Layout6D.layout6d - 5APC4100_TGL2_000/mapp6D/Layout6D.layout6d
```
Element Layout6D_Big (Type=layout6d)
  GridSize = 0
  UserOrigin:
    OffsetX = 0
    OffsetY = 0
  Segments:
    SegRow = 20
    SegCol = 4
    Segment[1]:
      TypeGrid240 = 0
      TypeGrid120 = 0
      TypeGrid320 = 0
      TypeGrid160 = 0
      X = 0
      Y = 0
      Name = Segment1
      IsMaster = TRUE
      PowerSectorName
      Gaps:
        Left = 0
        Bottom = 0
        Right = 0
        Top = 0
        S4Left = 0
        S4Bottom = 0
        S4Right = 0
        S4Top = 0
      BorderID:
        Left = 0
        Bottom = 0
        Right = 0
        Top = 0
    Segment[2]:
      TypeGrid240 = 0
      TypeGrid120 = 0
      TypeGrid320 = 0
      TypeGrid160 = 0
      X = 0
      Y = 1
      Name = Segment2
      IsMaster = false
      PowerSectorName
      Gaps:
        Left = 0
        Bottom = 0
        Right = 0
        Top = 0
        S4Left = 0
        S4Bottom = 0
        S4Right = 0
        S4Top = 0
      BorderID:
        Left = 0
        Bottom = 0
        Right = 0
        Top = 0
    Segment[3]:
      TypeGrid240 = 0
      TypeGrid120 = 0
      TypeGrid320 = 0
      TypeGrid160 = 0
      X = 0
      Y = 6
      Name = Segment3
      IsMaster = false
      PowerSectorName
      Gaps:
        Left = 0
        Bottom = 0
        Right = 0
        Top = 0
        S4Left = 0
        S4Bottom = 0
        S4Right = 0
        S4Top = 0
      BorderID:
        Left = 0
        Bottom = 0
        Right = 0
        Top = 0
    Segment[4]:
      TypeGrid240 = 0
      TypeGrid120 = 0
      TypeGrid320 = 0
      TypeGrid160 = 0
      X = 0
      Y = 7
      Name = Segment4
      IsMaster = false
      PowerSectorName
      Gaps:
        Left = 0
        Bottom = 0
        Right = 0
        Top = 0
        S4Left = 0
        S4Bottom = 0
        S4Right = 0
        S4Top = 0
      BorderID:
        Left = 0
        Bottom = 0
        Right = 0
        Top = 0
    Segment[5]:
      TypeGrid240 = 0
      TypeGrid120 = 0
      TypeGrid320 = 0
      TypeGrid160 = 0
      X = 0
      Y = 12
      Name = Segment5
      IsMaster = false
      PowerSectorName
      Gaps:
        Left = 0
        Bottom = 0
        Right = 0
        Top = 0
        S4Left = 0
        S4Bottom = 0
        S4Right = 0
        S4Top = 0
      BorderID:
        Left = 0
        Bottom = 0
        Right = 0
        Top = 0
    Segment[6]:
      TypeGrid240 = 0
      TypeGrid120 = 0
      TypeGrid320 = 0
      TypeGrid160 = 0
      X = 0
      Y = 13
      Name = Segment6
      IsMaster = false
      PowerSectorName
      Gaps:
        Left = 0
        Bottom = 0
        Right = 0
        Top = 0
        S4Left = 0
        S4Bottom = 0
        S4Right = 0
        S4Top = 0
      BorderID:
        Left = 0
        Bottom = 0
        Right = 0
        Top = 0
    Segment[7]:
      TypeGrid240 = 0
      TypeGrid120 = 0
      TypeGrid320 = 0
      TypeGrid160 = 0
      X = 0
      Y = 18
      Name = Segment7
      IsMaster = false
      PowerSectorName
      Gaps:
        Left = 0
        Bottom = 0
        Right = 0
        Top = 0
        S4Left = 0
        S4Bottom = 0
        S4Right = 0
        S4Top = 0
      BorderID:
        Left = 0
        Bottom = 0
        Right = 0
        Top = 0
    Segment[8]:
      TypeGrid240 = 0
      TypeGrid120 = 0
      TypeGrid320 = 0
      TypeGrid160 = 0
      X = 0
      Y = 19
      Name = Segment8
      IsMaster = false
      PowerSectorName
      Gaps:
        Left = 0
        Bottom = 0
        Right = 0
        Top = 0
        S4Left = 0
        S4Bottom = 0
        S4Right = 0
        S4Top = 0
      BorderID:
        Left = 0
        Bottom = 0
        Right = 0
        Top = 0
    Segment[9]:
      TypeGrid240 = 0
      TypeGrid120 = 0
      TypeGrid320 = 0
      TypeGrid160 = 0
      X = 1
      Y = 0
      Name = Segment9
      IsMaster = false
      PowerSectorName
      Gaps:
        Left = 0
        Bottom = 0
        Right = 0
        Top = 0
        S4Left = 0
        S4Bottom = 0
        S4Right = 0
        S4Top = 0
      BorderID:
        Left = 0
        Bottom = 0
        Right = 0
        Top = 0
    Segment[10]:
      TypeGrid240 = 0
      TypeGrid120 = 0
      TypeGrid320 = 0
      TypeGrid160 = 0
      X = 1
      Y = 1
      Name = Segment10
      IsMaster = false
      PowerSectorName
      Gaps:
        Left = 0
        Bottom = 0
        Right = 0
        Top = 0
        S4Left = 0
        S4Bottom = 0
        S4Right = 0
        S4Top = 0
      BorderID:
        Left = 0
        Bottom = 0
        Right = 0
        Top = 0
    Segment[11]:
      TypeGrid240 = 0
      TypeGrid120 = 0
      TypeGrid320 = 0
      TypeGrid160 = 0
      X = 1
      Y = 2
      Name = Segment11
      IsMaster = false
      PowerSectorName
      Gaps:
        Left = 0
        Bottom = 0
        Right = 0
        Top = 0
        S4Left = 0
        S4Bottom = 0
        S4Right = 0
        S4Top = 0
      BorderID:
        Left = 0
        Bottom = 0
        Right = 0
        Top = 0
    Segment[12]:
      TypeGrid240 = 0
      TypeGrid120 = 0
      TypeGrid320 = 0
      TypeGrid160 = 0
      X = 1
      Y = 3
      Name = Segment12
      IsMaster = false
      PowerSectorName
      Gaps:
        Left = 0
        Bottom = 0
        Right = 0
        Top = 0
        S4Left = 0
        S4Bottom = 0
        S4Right = 0
        S4Top = 0
      BorderID:
        Left = 0
        Bottom = 0
        Right = 0
        Top = 0
    Segment[13]:
      TypeGrid240 = 0
      TypeGrid120 = 0
      TypeGrid320 = 0
      TypeGrid160 = 0
      X = 1
      Y = 4
      Name = Segment13
      IsMaster = false
      PowerSectorName
      Gaps:
        Left = 0
        Bottom = 0
        Right = 0
        Top = 0
        S4Left = 0
        S4Bottom = 0
        S4Right = 0
        S4Top = 0
      BorderID:
        Left = 0
        Bottom = 0
        Right = 0
        Top = 0
    Segment[14]:
      TypeGrid240 = 0
      TypeGrid120 = 0
      TypeGrid320 = 0
      TypeGrid160 = 0
      X = 1
      Y = 5
      Name = Segment14
      IsMaster = false
      PowerSectorName
      Gaps:
        Left = 0
        Bottom = 0
        Right = 0
        Top = 0
        S4Left = 0
        S4Bottom = 0
        S4Right = 0
        S4Top = 0
      BorderID:
        Left = 0
        Bottom = 0
        Right = 0
        Top = 0
    Segment[15]:
      TypeGrid240 = 0
      TypeGrid120 = 0
      TypeGrid320 = 0
      TypeGrid160 = 0
      X = 1
      Y = 6
      Name = Segment15
      IsMaster = false
      PowerSectorName
      Gaps:
        Left = 0
        Bottom = 0
        Right = 0
        Top = 0
        S4Left = 0
        S4Bottom = 0
        S4Right = 0
        S4Top = 0
      BorderID:
        Left = 0
        Bottom = 0
        Right = 0
        Top = 0
    Segment[16]:
      TypeGrid240 = 0
      TypeGrid120 = 0
      TypeGrid320 = 0
      TypeGrid160 = 0
      X = 1
      Y = 7
      Name = Segment16
      IsMaster = false
      PowerSectorName
      Gaps:
        Left = 0
        Bottom = 0
        Right = 0
        Top = 0
        S4Left = 0
        S4Bottom = 0
        S4Right = 0
        S4Top = 0
      BorderID:
        Left = 0
        Bottom = 0
        Right = 0
        Top = 0
    Segment[17]:
      TypeGrid240 = 0
      TypeGrid120 = 0
      TypeGrid320 = 0
      TypeGrid160 = 0
      X = 1
      Y = 8
      Name = Segment17
      IsMaster = false
      PowerSectorName
      Gaps:
        Left = 0
        Bottom = 0
        Right = 0
        Top = 0
        S4Left = 0
        S4Bottom = 0
        S4Right = 0
        S4Top = 0
      BorderID:
        Left = 0
        Bottom = 0
        Right = 0
        Top = 0
    Segment[18]:
      TypeGrid240 = 0
      TypeGrid120 = 0
      TypeGrid320 = 0
      TypeGrid160 = 0
      X = 1
      Y = 9
      Name = Segment18
      IsMaster = false
      PowerSectorName
      Gaps:
        Left = 0
        Bottom = 0
        Right = 0
        Top = 0
        S4Left = 0
        S4Bottom = 0
        S4Right = 0
        S4Top = 0
      BorderID:
        Left = 0
        Bottom = 0
        Right = 0
        Top = 0
    Segment[19]:
      TypeGrid240 = 0
      TypeGrid120 = 0
      TypeGrid320 = 0
      TypeGrid160 = 0
      X = 1
      Y = 10
      Name = Segment19
      IsMaster = false
      PowerSectorName
      Gaps:
        Left = 0
        Bottom = 0
        Right = 0
        Top = 0
        S4Left = 0
        S4Bottom = 0
        S4Right = 0
        S4Top = 0
      BorderID:
        Left = 0
        Bottom = 0
        Right = 0
        Top = 0
    Segment[20]:
      TypeGrid240 = 0
      TypeGrid120 = 0
      TypeGrid320 = 0
      TypeGrid160 = 0
      X = 1
      Y = 11
      Name = Segment20
      IsMaster = false
      PowerSectorName
      Gaps:
        Left = 0
        Bottom = 0
        Right = 0
        Top = 0
        S4Left = 0
        S4Bottom = 0
        S4Right = 0
        S4Top = 0
      BorderID:
        Left = 0
        Bottom = 0
        Right = 0
        Top = 0
    Segment[21]:
      TypeGrid240 = 0
      TypeGrid120 = 0
      TypeGrid320 = 0
      TypeGrid160 = 0
      X = 1
      Y = 12
      Name = Segment21
      IsMaster = false
      PowerSectorName
      Gaps:
        Left = 0
        Bottom = 0
        Right = 0
        Top = 0
        S4Left = 0
        S4Bottom = 0
        S4Right = 0
        S4Top = 0
      BorderID:
        Left = 0
        Bottom = 0
        Right = 0
        Top = 0
    Segment[22]:
      TypeGrid240 = 0
      TypeGrid120 = 0
      TypeGrid320 = 0
      TypeGrid160 = 0
      X = 1
      Y = 13
      Name = Segment22
      IsMaster = false
      PowerSectorName
      Gaps:
        Left = 0
        Bottom = 0
        Right = 0
        Top = 0
        S4Left = 0
        S4Bottom = 0
        S4Right = 0
        S4Top = 0
      BorderID:
        Left = 0
        Bottom = 0
        Right = 0
        Top = 0
    Segment[23]:
      TypeGrid240 = 0
      TypeGrid120 = 0
      TypeGrid320 = 0
      TypeGrid160 = 0
      X = 1
      Y = 14
      Name = Segment23
      IsMaster = false
      PowerSectorName
      Gaps:
        Left = 0
        Bottom = 0
        Right = 0
        Top = 0
        S4Left = 0
        S4Bottom = 0
        S4Right = 0
        S4Top = 0
      BorderID:
        Left = 0
        Bottom = 0
        Right = 0
        Top = 0
    Segment[24]:
      TypeGrid240 = 0
      TypeGrid120 = 0
      TypeGrid320 = 0
      TypeGrid160 = 0
      X = 1
      Y = 15
      Name = Segment24
      IsMaster = false
      PowerSectorName
      Gaps:
        Left = 0
        Bottom = 0
        Right = 0
        Top = 0
        S4Left = 0
        S4Bottom = 0
        S4Right = 0
        S4Top = 0
      BorderID:
        Left = 0
        Bottom = 0
        Right = 0
        Top = 0
    Segment[25]:
      TypeGrid240 = 0
      TypeGrid120 = 0
      TypeGrid320 = 0
      TypeGrid160 = 0
      X = 1
      Y = 16
      Name = Segment25
      IsMaster = false
      PowerSectorName
      Gaps:
        Left = 0
        Bottom = 0
        Right = 0
        Top = 0
        S4Left = 0
        S4Bottom = 0
        S4Right = 0
        S4Top = 0
      BorderID:
        Left = 0
        Bottom = 0
        Right = 0
        Top = 0
    Segment[26]:
      TypeGrid240 = 0
      TypeGrid120 = 0
      TypeGrid320 = 0
      TypeGrid160 = 0
      X = 1
      Y = 17
      Name = Segment26
      IsMaster = false
      PowerSectorName
      Gaps:
        Left = 0
        Bottom = 0
        Right = 0
        Top = 0
        S4Left = 0
        S4Bottom = 0
        S4Right = 0
        S4Top = 0
      BorderID:
        Left = 0
        Bottom = 0
        Right = 0
        Top = 0
    Segment[27]:
      TypeGrid240 = 0
      TypeGrid120 = 0
      TypeGrid320 = 0
      TypeGrid160 = 0
      X = 1
      Y = 18
      Name = Segment27
      IsMaster = false
      PowerSectorName
      Gaps:
        Left = 0
        Bottom = 0
        Right = 0
        Top = 0
        S4Left = 0
        S4Bottom = 0
        S4Right = 0
        S4Top = 0
      BorderID:
        Left = 0
        Bottom = 0
        Right = 0
        Top = 0
    Segment[28]:
      TypeGrid240 = 0
      TypeGrid120 = 0
      TypeGrid320 = 0
      TypeGrid160 = 0
      X = 1
      Y = 19
      Name = Segment28
      IsMaster = false
      PowerSectorName
      Gaps:
        Left = 0
        Bottom = 0
        Right = 0
        Top = 0
        S4Left = 0
        S4Bottom = 0
        S4Right = 0
        S4Top = 0
      BorderID:
        Left = 0
        Bottom = 0
        Right = 0
        Top = 0
    Segment[29]:
      TypeGrid240 = 0
      TypeGrid120 = 0
      TypeGrid320 = 0
      TypeGrid160 = 0
      X = 2
      Y = 0
      Name = Segment29
      IsMaster = false
      PowerSectorName
      Gaps:
        Left = 0
        Bottom = 0
        Right = 0
        Top = 0
        S4Left = 0
        S4Bottom = 0
        S4Right = 0
        S4Top = 0
      BorderID:
        Left = 0
        Bottom = 0
        Right = 0
        Top = 0
    Segment[30]:
      TypeGrid240 = 0
      TypeGrid120 = 0
      TypeGrid320 = 0
      TypeGrid160 = 0
      X = 2
      Y = 1
      Name = Segment30
      IsMaster = false
      PowerSectorName
      Gaps:
        Left = 0
        Bottom = 0
        Right = 0
        Top = 0
        S4Left = 0
        S4Bottom = 0
        S4Right = 0
        S4Top = 0
      BorderID:
        Left = 0
        Bottom = 0
        Right = 0
        Top = 0
    Segment[31]:
      TypeGrid240 = 0
      TypeGrid120 = 0
      TypeGrid320 = 0
      TypeGrid160 = 0
      X = 2
      Y = 2
      Name = Segment31
      IsMaster = false
      PowerSectorName
      Gaps:
        Left = 0
        Bottom = 0
        Right = 0
        Top = 0
        S4Left = 0
        S4Bottom = 0
        S4Right = 0
        S4Top = 0
      BorderID:
        Left = 0
        Bottom = 0
        Right = 0
        Top = 0
    Segment[32]:
      TypeGrid240 = 0
      TypeGrid120 = 0
      TypeGrid320 = 0
      TypeGrid160 = 0
      X = 2
      Y = 3
      Name = Segment32
      IsMaster = false
      PowerSectorName
      Gaps:
        Left = 0
        Bottom = 0
        Right = 0
        Top = 0
        S4Left = 0
        S4Bottom = 0
        S4Right = 0
        S4Top = 0
      BorderID:
        Left = 0
        Bottom = 0
        Right = 0
        Top = 0
    Segment[33]:
      TypeGrid240 = 0
      TypeGrid120 = 0
      TypeGrid320 = 0
      TypeGrid160 = 0
      X = 2
      Y = 4
      Name = Segment33
      IsMaster = false
      PowerSectorName
      Gaps:
        Left = 0
        Bottom = 0
        Right = 0
        Top = 0
        S4Left = 0
        S4Bottom = 0
        S4Right = 0
        S4Top = 0
      BorderID:
        Left = 0
        Bottom = 0
        Right = 0
        Top = 0
    Segment[34]:
      TypeGrid240 = 0
      TypeGrid120 = 0
      TypeGrid320 = 0
      TypeGrid160 = 0
      X = 2
      Y = 5
      Name = Segment34
      IsMaster = false
      PowerSectorName
      Gaps:
        Left = 0
        Bottom = 0
        Right = 0
        Top = 0
        S4Left = 0
        S4Bottom = 0
        S4Right = 0
        S4Top = 0
      BorderID:
        Left = 0
        Bottom = 0
        Right = 0
        Top = 0
    Segment[35]:
      TypeGrid240 = 0
      TypeGrid120 = 0
      TypeGrid320 = 0
      TypeGrid160 = 0
      X = 2
      Y = 6
      Name = Segment35
      IsMaster = false
      PowerSectorName
      Gaps:
        Left = 0
        Bottom = 0
        Right = 0
        Top = 0
        S4Left = 0
        S4Bottom = 0
        S4Right = 0
        S4Top = 0
      BorderID:
        Left = 0
        Bottom = 0
        Right = 0
        Top = 0
    Segment[36]:
      TypeGrid240 = 0
      TypeGrid120 = 0
      TypeGrid320 = 0
      TypeGrid160 = 0
      X = 2
      Y = 7
      Name = Segment36
      IsMaster = false
      PowerSectorName
      Gaps:
        Left = 0
        Bottom = 0
        Right = 0
        Top = 0
        S4Left = 0
        S4Bottom = 0
        S4Right = 0
        S4Top = 0
      BorderID:
        Left = 0
        Bottom = 0
        Right = 0
        Top = 0
    Segment[37]:
      TypeGrid240 = 0
      TypeGrid120 = 0
      TypeGrid320 = 0
      TypeGrid160 = 0
      X = 2
      Y = 8
      Name = Segment37
      IsMaster = false
      PowerSectorName
      Gaps:
        Left = 0
        Bottom = 0
        Right = 0
        Top = 0
        S4Left = 0
        S4Bottom = 0
        S4Right = 0
        S4Top = 0
      BorderID:
        Left = 0
        Bottom = 0
        Right = 0
        Top = 0
    Segment[38]:
      TypeGrid240 = 0
      TypeGrid120 = 0
      TypeGrid320 = 0
      TypeGrid160 = 0
      X = 2
      Y = 9
      Name = Segment38
      IsMaster = false
      PowerSectorName
      Gaps:
        Left = 0
        Bottom = 0
        Right = 0
        Top = 0
        S4Left = 0
        S4Bottom = 0
        S4Right = 0
        S4Top = 0
      BorderID:
        Left = 0
        Bottom = 0
        Right = 0
        Top = 0
    Segment[39]:
      TypeGrid240 = 0
      TypeGrid120 = 0
      TypeGrid320 = 0
      TypeGrid160 = 0
      X = 2
      Y = 10
      Name = Segment39
      IsMaster = false
      PowerSectorName
      Gaps:
        Left = 0
        Bottom = 0
        Right = 0
        Top = 0
        S4Left = 0
        S4Bottom = 0
        S4Right = 0
        S4Top = 0
      BorderID:
        Left = 0
        Bottom = 0
        Right = 0
        Top = 0
    Segment[40]:
      TypeGrid240 = 0
      TypeGrid120 = 0
      TypeGrid320 = 0
      TypeGrid160 = 0
      X = 2
      Y = 11
      Name = Segment40
      IsMaster = false
      PowerSectorName
      Gaps:
        Left = 0
        Bottom = 0
        Right = 0
        Top = 0
        S4Left = 0
        S4Bottom = 0
        S4Right = 0
        S4Top = 0
      BorderID:
        Left = 0
        Bottom = 0
        Right = 0
        Top = 0
    Segment[41]:
      TypeGrid240 = 0
      TypeGrid120 = 0
      TypeGrid320 = 0
      TypeGrid160 = 0
      X = 2
      Y = 12
      Name = Segment41
      IsMaster = false
      PowerSectorName
      Gaps:
        Left = 0
        Bottom = 0
        Right = 0
        Top = 0
        S4Left = 0
        S4Bottom = 0
        S4Right = 0
        S4Top = 0
      BorderID:
        Left = 0
        Bottom = 0
        Right = 0
        Top = 0
    Segment[42]:
      TypeGrid240 = 0
      TypeGrid120 = 0
      TypeGrid320 = 0
      TypeGrid160 = 0
      X = 2
      Y = 13
      Name = Segment42
      IsMaster = false
      PowerSectorName
      Gaps:
        Left = 0
        Bottom = 0
        Right = 0
        Top = 0
        S4Left = 0
        S4Bottom = 0
        S4Right = 0
        S4Top = 0
      BorderID:
        Left = 0
        Bottom = 0
        Right = 0
        Top = 0
    Segment[43]:
      TypeGrid240 = 0
      TypeGrid120 = 0
      TypeGrid320 = 0
      TypeGrid160 = 0
      X = 2
      Y = 14
      Name = Segment43
      IsMaster = false
      PowerSectorName
      Gaps:
        Left = 0
        Bottom = 0
        Right = 0
        Top = 0
        S4Left = 0
        S4Bottom = 0
        S4Right = 0
        S4Top = 0
      BorderID:
        Left = 0
        Bottom = 0
        Right = 0
        Top = 0
    Segment[44]:
      TypeGrid240 = 0
      TypeGrid120 = 0
      TypeGrid320 = 0
      TypeGrid160 = 0
      X = 2
      Y = 15
      Name = Segment44
      IsMaster = false
      PowerSectorName
      Gaps:
        Left = 0
        Bottom = 0
        Right = 0
        Top = 0
        S4Left = 0
        S4Bottom = 0
        S4Right = 0
        S4Top = 0
      BorderID:
        Left = 0
        Bottom = 0
        Right = 0
        Top = 0
    Segment[45]:
      TypeGrid240 = 0
      TypeGrid120 = 0
      TypeGrid320 = 0
      TypeGrid160 = 0
      X = 2
      Y = 16
      Name = Segment45
      IsMaster = false
      PowerSectorName
      Gaps:
        Left = 0
        Bottom = 0
        Right = 0
        Top = 0
        S4Left = 0
        S4Bottom = 0
        S4Right = 0
        S4Top = 0
      BorderID:
        Left = 0
        Bottom = 0
        Right = 0
        Top = 0
    Segment[46]:
      TypeGrid240 = 0
      TypeGrid120 = 0
      TypeGrid320 = 0
      TypeGrid160 = 0
      X = 2
      Y = 17
      Name = Segment46
      IsMaster = false
      PowerSectorName
      Gaps:
        Left = 0
        Bottom = 0
        Right = 0
        Top = 0
        S4Left = 0
        S4Bottom = 0
        S4Right = 0
        S4Top = 0
      BorderID:
        Left = 0
        Bottom = 0
        Right = 0
        Top = 0
    Segment[47]:
      TypeGrid240 = 0
      TypeGrid120 = 0
      TypeGrid320 = 0
      TypeGrid160 = 0
      X = 2
      Y = 18
      Name = Segment47
      IsMaster = false
      PowerSectorName
      Gaps:
        Left = 0
        Bottom = 0
        Right = 0
        Top = 0
        S4Left = 0
        S4Bottom = 0
        S4Right = 0
        S4Top = 0
      BorderID:
        Left = 0
        Bottom = 0
        Right = 0
        Top = 0
    Segment[48]:
      TypeGrid240 = 0
      TypeGrid120 = 0
      TypeGrid320 = 0
      TypeGrid160 = 0
      X = 2
      Y = 19
      Name = Segment48
      IsMaster = false
      PowerSectorName
      Gaps:
        Left = 0
        Bottom = 0
        Right = 0
        Top = 0
        S4Left = 0
        S4Bottom = 0
        S4Right = 0
        S4Top = 0
      BorderID:
        Left = 0
        Bottom = 0
        Right = 0
        Top = 0
    Segment[49]:
      TypeGrid240 = 0
      TypeGrid120 = 0
      TypeGrid320 = 0
      TypeGrid160 = 0
      X = 3
      Y = 0
      Name = Segment49
      IsMaster = false
      PowerSectorName
      Gaps:
        Left = 0
        Bottom = 0
        Right = 0
        Top = 0
        S4Left = 0
        S4Bottom = 0
        S4Right = 0
        S4Top = 0
      BorderID:
        Left = 0
        Bottom = 0
        Right = 0
        Top = 0
    Segment[50]:
      TypeGrid240 = 0
      TypeGrid120 = 0
      TypeGrid320 = 0
      TypeGrid160 = 0
      X = 3
      Y = 1
      Name = Segment50
      IsMaster = false
      PowerSectorName
      Gaps:
        Left = 0
        Bottom = 0
        Right = 0
        Top = 0
        S4Left = 0
        S4Bottom = 0
        S4Right = 0
        S4Top = 0
      BorderID:
        Left = 0
        Bottom = 0
        Right = 0
        Top = 0
    Segment[51]:
      TypeGrid240 = 0
      TypeGrid120 = 0
      TypeGrid320 = 0
      TypeGrid160 = 0
      X = 3
      Y = 6
      Name = Segment51
      IsMaster = false
      PowerSectorName
      Gaps:
        Left = 0
        Bottom = 0
        Right = 0
        Top = 0
        S4Left = 0
        S4Bottom = 0
        S4Right = 0
        S4Top = 0
      BorderID:
        Left = 0
        Bottom = 0
        Right = 0
        Top = 0
    Segment[52]:
      TypeGrid240 = 0
      TypeGrid120 = 0
      TypeGrid320 = 0
      TypeGrid160 = 0
      X = 3
      Y = 7
      Name = Segment52
      IsMaster = false
      PowerSectorName
      Gaps:
        Left = 0
        Bottom = 0
        Right = 0
        Top = 0
        S4Left = 0
        S4Bottom = 0
        S4Right = 0
        S4Top = 0
      BorderID:
        Left = 0
        Bottom = 0
        Right = 0
        Top = 0
    Segment[53]:
      TypeGrid240 = 0
      TypeGrid120 = 0
      TypeGrid320 = 0
      TypeGrid160 = 0
      X = 3
      Y = 12
      Name = Segment53
      IsMaster = false
      PowerSectorName
      Gaps:
        Left = 0
        Bottom = 0
        Right = 0
        Top = 0
        S4Left = 0
        S4Bottom = 0
        S4Right = 0
        S4Top = 0
      BorderID:
        Left = 0
        Bottom = 0
        Right = 0
        Top = 0
    Segment[54]:
      TypeGrid240 = 0
      TypeGrid120 = 0
      TypeGrid320 = 0
      TypeGrid160 = 0
      X = 3
      Y = 13
      Name = Segment54
      IsMaster = false
      PowerSectorName
      Gaps:
        Left = 0
        Bottom = 0
        Right = 0
        Top = 0
        S4Left = 0
        S4Bottom = 0
        S4Right = 0
        S4Top = 0
      BorderID:
        Left = 0
        Bottom = 0
        Right = 0
        Top = 0
    Segment[55]:
      TypeGrid240 = 0
      TypeGrid120 = 0
      TypeGrid320 = 0
      TypeGrid160 = 0
      X = 3
      Y = 18
      Name = Segment55
      IsMaster = false
      PowerSectorName
      Gaps:
        Left = 0
        Bottom = 0
        Right = 0
        Top = 0
        S4Left = 0
        S4Bottom = 0
        S4Right = 0
        S4Top = 0
      BorderID:
        Left = 0
        Bottom = 0
        Right = 0
        Top = 0
    Segment[56]:
      TypeGrid240 = 0
      TypeGrid120 = 0
      TypeGrid320 = 0
      TypeGrid160 = 0
      X = 3
      Y = 19
      Name = Segment56
      IsMaster = false
      PowerSectorName
      Gaps:
        Left = 0
        Bottom = 0
        Right = 0
        Top = 0
        S4Left = 0
        S4Bottom = 0
        S4Right = 0
        S4Top = 0
      BorderID:
        Left = 0
        Bottom = 0
        Right = 0
        Top = 0
  Synchronization = NotUsed
```

### Config.mappconnect - 5APC4100_TGL2_000/mappConnect/Config.mappconnect
```
Element mapp Connect Configuration (Type=mappconnect)
  WebServerProtocol = 1
    WebServerPort = 8080
    Interface = All
    WebServerPortSsl = 8443
  WebServerEndpointConfiguration:
    Endpoint[1]:
      Endpoint = /*
      Roles
  OpcUaServerWhitelist:
    OpcUaServer[1]:
      Url = opc.tcp://127.0.0.1:4840
```

## Configuration Small

CPU 5APC4100.TGL2-000, AutomationRuntime 6.3.3, Build 11.3.0, Vc 6.0.0

### Task classes (Cpu.sw)
```
Cyclic#3:
  FirstProgr <- obsolete.FirstProgram.prg
NcDataObjects: McDriveLog
Binaries: FWRules, ArSvcReg, TCData, udbdef, McAcpDrv, iomap, Config_1, BRRole, arconfig, asfw, ashwac, sysconf, UaCsConfig, ashwd, Config_2, mvLoader
Libraries: AsZip, UaCoalPrv, runtime, astime, fileio, UaCoal, sys_lib, powerlnk, AsEPL, AsIecCon, AsBrMath, McAcp6DSys, ArSsl, AsBrStr, MpBase
```

### Hardware
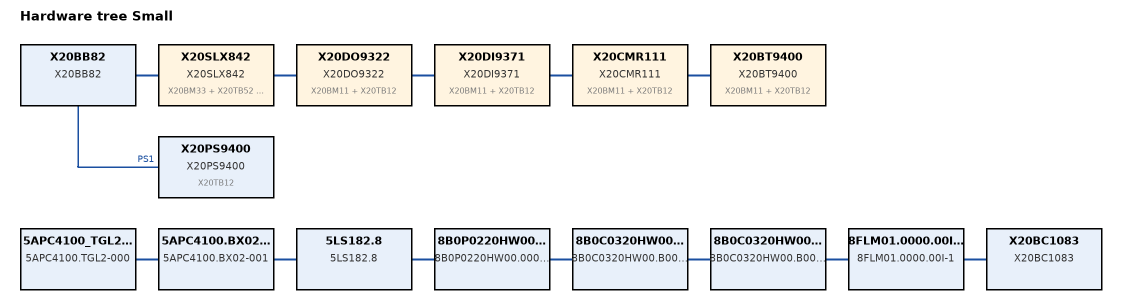
```
5APC4100.BX02-001 : 5APC4100.BX02-001 v1.0.0.0  [SY -> 5APC4100_TGL2_000.SY3]
5APC4100_TGL2_000 : 5APC4100.TGL2-000 v1.3.1.0
  Connector IF3:
    AssignedOperatingSystem = ARemb
    ActivateDevice = 1
    Mode = Manual
    InternetAddress = 192.168.1.201
    SubnetMask = 255.255.255.0
    ActivateSnmp = 2
  Connector IF4:
    AssignedOperatingSystem = ARemb
    ActivateDevice = 1
  Connector IF5:
    AssignedOperatingSystem = GPOS
  Connector IF6:
    AssignedOperatingSystem = GPOS
  Connector IF13:
    OperatingSystem = ARemb
    ActivateDevice = 1
  Connector IF7:
    AssignedOperatingSystem = GPOS
  Connector IF8:
    AssignedOperatingSystem = GPOS
  Connector IF9:
    AssignedOperatingSystem = GPOS
  Connector IF10:
    AssignedOperatingSystem = GPOS
  Connector IF11:
    AssignedOperatingSystem = ARemb
  Connector IF12:
    AssignedOperatingSystem = ARemb
  ConfigurationID = BothSystems_SmallSystem
  TimerDeviceType = EPLX2X
  TimerDevice = 5LS182.8.IF1
  TaskClassIdleTime = 2000
  Cyclic1Duration = 2000
  Cyclic1Tolerance = 0
  FileDevice1
  FileDeviceName1 = 6DData
  FileDevicePath1 = USER_PATH
  ActivateFtpServer = 1
  FTPProtocol = 1
  FtpUser1
  FtpUsername1 = admin
  FtpUserPassword1 = U6LVhgEhxdExLCAl9+GafDrOE8FUGhRIwZtJz/YbLrc=
  FtpUserSalt1 = 45uvzRU9
  FTPAccessRight1 = 0
  FTPdevice1 = ALL
  ActivateWebServer = 1
  ActivateSdm = 1
  ActivateHypervisor = 1
  ARembDramSizeInMb = 2048
5LS182.8 : 5LS182.8 v1.4.3.0  [SL -> 5APC4100.BX02-001.SL1]
8B0C0320HW00.B00-1_A : 8B0C0320HW00.B00-1 v1.0.1.3 (NodeNumber=3)  [PLK1 -> 8B0P0220HW00.000-1.PLK2 [Cable Type=PowerlinkCable, Length=10, Version=1.0.0.3]; PLK2 -> 8B0C0320HW00.B00-1_B.PLK1 [Cable Type=PowerlinkCable, Length=10, Version=1.0.0.3]]
  FunctionModel/PowerSection:
    AxisReference = A
8B0C0320HW00.B00-1_B : 8B0C0320HW00.B00-1 v1.0.1.3 (NodeNumber=4)  [PLK1 -> 8B0C0320HW00.B00-1_A.PLK2 [Cable Type=PowerlinkCable, Length=10, Version=1.0.0.3]; PLK2 -> 8FLM01.0000.00I-1.PLK1 [Cable Type=PowerlinkCable, Length=10, Version=1.0.0.3]]
  FunctionModel/PowerSection:
    AxisReference = B
8B0P0220HW00.000-1 : 8B0P0220HW00.000-1 v2.3.0.3 (NodeNumber=2)  [PLK1 -> 5LS182.8.IF1 [Cable Type=PowerlinkCable, Length=10, Version=1.0.0.3]; PLK2 -> 8B0C0320HW00.B00-1_A.PLK1 [Cable Type=PowerlinkCable, Length=10, Version=1.0.0.3]]
8FLM01.0000.00I-1 : 8FLM01.0000.00I-1 v1.0.0.2 (NodeNumber=239)  [PLK1 -> 8B0C0320HW00.B00-1_B.PLK2 [Cable Type=PowerlinkCable, Length=10, Version=1.0.0.3]; PLK2 -> X20BC1083.PLK1 [Cable Type=PowerlinkCable, Length=10, Version=1.0.0.3]]
  Supervision = off
X20BB82 : X20BB82 v1.2.0.0
X20BC1083 : X20BC1083 v2.16.1.0 (NodeNumber=1)  [PLK1 -> 8FLM01.0000.00I-1.PLK2 [Cable Type=PowerlinkCable, Length=10, Version=1.0.0.3]; SL -> X20BB82.SL1]
X20BM11 : X20BM11 v1.1.0.0  [X2X1 -> X20BM11_b.X2X2]
X20BM11_a : X20BM11 v1.1.0.0  [X2X1 -> X20BM33.X2X2]
X20BM11_b : X20BM11 v1.1.0.0  [X2X1 -> X20BM11_a.X2X2]
X20BM11_c : X20BM11 v1.1.0.0  [X2X1 -> X20BM11.X2X2]
X20BM33 : X20BM33 v1.1.0.0 (Disabled=true)  [X2X1 -> X20BB82.IF1]
X20BT9400 : X20BT9400 v1.3.1.0  [SS1 -> X20TB12_d.SS; SL -> X20BM11_c.SL1]
X20CMR111 : X20CMR111 v1.7.0.0  [SS1 -> X20TB12_a.SS; SL -> X20BM11.SL1]
X20DI9371 : X20DI9371 v1.6.1.0  [SS1 -> X20TB12_c.SS; SL -> X20BM11_b.SL1]
X20DO9322 : X20DO9322 v1.6.2.0  [SS1 -> X20TB12_b.SS; SL -> X20BM11_a.SL1]
X20PS9400 : X20PS9400 v1.8.1.0  [SS1 -> X20TB12.SS; PS -> X20BB82.PS1]
X20SLX842 : X20SLX842 v2.6.0.2 (Disabled=true)  [SS1 -> X20TB52.SS; SS2 -> X20TB52_a.SS; SL -> X20BM33.SL1]
X20TB12 : X20TB12 v1.0.0.0
X20TB12_a : X20TB12 v1.0.0.0
X20TB12_b : X20TB12 v1.0.0.0
X20TB12_c : X20TB12 v1.0.0.0
X20TB12_d : X20TB12 v1.0.0.0
X20TB52 : X20TB52 v1.0.0.2 (Disabled=true)
X20TB52_a : X20TB52 v1.0.0.2 (Disabled=true)
```
